                   6:  (* order finished *)
                       IF #sRecv.Echo.Start AND #sRecv.ErrorCode <> 16#FFFF THEN
                           #sSend.Start := FALSE;
                           #sHelp.EnableTime := FALSE;
                           IF #sRecv.ErrorCode = 16#0000 THEN
                               #sHelp.Step[#tIndex] := #sHelp.Step[#tIndex] + 1;
                           ELSE
                               #oErrorCode := 203;
                               #sHelp.Step[#tIndex] := 698;
                           END_IF;
                       ELSIF #sHelp.Abort THEN
                           #sHelp.Step[#tIndex] := 10;
                       ELSE
                           #sHelp.EnableTime := TRUE;
                           IF #sHelp.CmdTimer.Q THEN
                               #oErrorCode := 204;
                               #sHelp.Step[#tIndex] := 699;
                           END_IF;
                       END_IF;

                   7:  (* start order *)
                       IF (#sRecv.Echo.Status = 16#0000) AND #sRecv.CycleEnd THEN
                           #sSend.ReadLastResult := TRUE;
                           #sHelp.EnableTime := FALSE;
                           #sHelp.Step[#tIndex] := #sHelp.Step[#tIndex] + 1;
                       END_IF;

                   8:  (* order accepted *)
                       IF #sRecv.Echo.ReadLastResult AND #sRecv.ErrorCode = 16#FFFF THEN
                           #sHelp.EnableTime := FALSE;
                           #sHelp.Step[#tIndex] := #sHelp.Step[#tIndex] + 1;
                       ELSE
                           #sHelp.EnableTime := TRUE;
                           IF #sHelp.CmdTimer.Q THEN
                               #oErrorCode := 204;
                               #sHelp.Step[#tIndex] := 899;
                           END_IF;
                       END_IF;

                   9:  (* order finished *)
                       IF #sRecv.Echo.ReadLastResult AND #sRecv.ErrorCode <> 16#FFFF THEN
                           #sSend.ReadLastResult := FALSE;
                           #sHelp.EnableTime := FALSE;
                           IF #sRecv.ErrorCode = 16#0000 THEN
                               #sHelp.Step[#tIndex] := 997;
                           ELSE
                               #oErrorCode := 203;
                               #sHelp.Step[#tIndex] := 998;
                           END_IF;
                       ELSE
                           #sHelp.EnableTime := TRUE;
                           IF #sHelp.CmdTimer.Q THEN
                               #oErrorCode := 204;
                               #sHelp.Step[#tIndex] := 999;
                           END_IF;
                       END_IF;

                   10:  (* abort order *)
                       #sHelp.Step[#tIndex] := 1099;

                   299,398,399,599,698,699,899,997,998,999,1099:
                       #sSend.Reset := FALSE;
                       #sSend.Start := FALSE;
                       #sSend.ReadLastResult := FALSE;
                       #sHelp.MeasureAct := FALSE;
                       #sHMI.Trigger.Measure := FALSE;
                       #sHelp.Abort := FALSE;
                       IF #oErrorCode = 0 THEN
                           #oResult := #sRecv.Result;
                           #oMeasureOk := TRUE;
                       END_IF;
               END_CASE;
           END_IF;
       END_REGION

       (* update outputs *)
       #oDeviceReady := #sRecv.CycleEnd;
       #oPressure.Value := UDINT_TO_REAL(#sRecv.ActPressure) / 1000.0;
       CASE #sRecv.PressureUnitCode OF
           0000:
               #oPressure.Unit := 'cm3/s';
           1000:
               #oPressure.Unit := 'cm3/min';
           2000:
               #oPressure.Unit := 'cm3/h';
           3000:
               #oPressure.Unit := 'mm3/h';
           4000:
               #oPressure.Unit := 'Pa';
           5000:
               #oPressure.Unit := 'Pa/s';
           6000:
               #oPressure.Unit := 'Pa';
           7000:
               #oPressure.Unit := 'Pa';
           8000:
               #oPressure.Unit := 'Pa/s';
           9000:
               #oPressure.Unit := 'Pa/s';
           11000:
               #oPressure.Unit := 'bar';
           12000:
               #oPressure.Unit := 'KPa';
           13000:
               #oPressure.Unit := 'psi';
           14000:
               #oPressure.Unit := 'mbar';
           15000:
               #oPressure.Unit := 'MPa';
           43000:
               #oPressure.Unit := 'Pa';
           44000:
               #oPressure.Unit := 'Pa';
           45000:
               #oPressure.Unit := 'Pa/s';
           46000:
               #oPressure.Unit := 'In3/s';
           47000:
               #oPressure.Unit := 'In3/min';
           48000:
               #oPressure.Unit := 'In3/h';
           49000:
               #oPressure.Unit := 'Ft3/h';
           50000:
               #oPressure.Unit := 'mL/s';
           51000:
               #oPressure.Unit := 'mL/min';
           52000:
               #oPressure.Unit := 'mL/h';
           58000:
               #oPressure.Unit := 'cm3/s';
           59000:
               #oPressure.Unit := 'cm3/min';
           60000:
               #oPressure.Unit := 'cm3/h';
           76000:
               #oPressure.Unit := 'Ft3/s';
           77000:
               #oPressure.Unit := 'Ft3/min';
           84000:
               #oPressure.Unit := 'sccm';
           ELSE
               ;
       END_CASE;
       #oActProgStep := #sRecv.ActProgStep;
       #oActProgNo := #sRecv.ActProgram + 1;

       (* update hmi *)
       #sHMI.Status.DeviceReady := #oDeviceReady;
       #sHMI.Status.Ready := #oReady;
       #sHMI.Status.Error := #oError;
       #sHMI.Status.SetProgOk := #oSetProgOk;
       #sHMI.Status.MeasureOk := #oMeasureOk;
       #sHMI.Status.ErrorCode := #oErrorCode;
       #sHMI.Status.Result := #oResult;
       #sHMI.Status.Pressure := #oPressure;
       #sHMI.Status.ActProgStep := #oActProgStep;
       #sHMI.Status.ActProgNo := #oActProgNo;
       #sHMI.Status.ElapsedTime := #oElapsedTime;

       (* set ready for command flag *)
       IF (#oErrorCode = 0) AND (#sHelp.OrderCnt = 0) AND #oDeviceReady AND NOT #sHelp.SetProgAct AND NOT #sHelp.MeasureAct THEN
           #oReady := TRUE;
       ELSE
           #oReady := FALSE;
       END_IF;

       (* move static bits to output bytes *)
       #sArrayOutput[1, 1].%X0 := #sSend.Reset;
       #sArrayOutput[1, 1].%X1 := #sSend.Start;
       #sArrayOutput[1, 1].%X2 := #sSend.StartSpec;
       #sArrayOutput[1, 1].%X3 := #sSend.ProgramSel AND "ClockMemory0.8s";
       #sArrayOutput[1, 1].%X5 := #sSend.ReadPara ;
       #sArrayOutput[1, 2].%X7 := #sSend.ReadLastResult AND "ClockMemory0.8s";
       #sArrayOutput[1, 7] := #sSend.ProgNo.%B0;
       REGION SpecialCycle
           // Statement section REGION
           IF NOT #ioSpecialCycle THEN
               #SpecialCycleStep := 0;
           END_IF;
           IF #ioSpecialCycle AND #SpecialCycleStep = 0 AND #oReady AND #oDeviceReady THEN
               #SpecialCycleStep := 10;
           END_IF;
           #IEC_Timer_0_Instance(IN := #SpecialCycleStep = 10,
                                 PT := t#0.2s);
           #IEC_Timer_1_Instance(IN := #SpecialCycleStep = 20,
                                 PT := t#0.4s);
           CASE #SpecialCycleStep OF
               10://标志清零
                   #sHelp.EnableTime := FALSE;
                   #sArrayOutput[1, 9] := 16#00;
                   #sArrayOutput[1, 10] := 16#00;
                   IF #IEC_Timer_0_Instance.Q THEN
                       #SpecialCycleStep := 20;
                   END_IF;
               20://赋值
                   #sHelp.EnableTime := FALSE;
                   #sArrayOutput[1, 9] := 16#08;
                   #sArrayOutput[1, 10] := 16#00;
                   #sSend.StartSpec := 1;
                   IF #IEC_Timer_1_Instance.Q THEN
                       #SpecialCycleStep := 30;
                   END_IF;

               30://触发
                   #sHelp.EnableTime := FALSE;
                   #sSend.Start := 1;
                   #SpecialCycleStep := 40;
               40://运行
                   IF #sRecv.Echo.StartSpec THEN
                       #sHelp.EnableTime := FALSE;
                       #SpecialCycleStep := 50;
                   END_IF;
                   #sHelp.EnableTime := TRUE;
                   IF #sHelp.CmdTimer.Q THEN
                       #oErrorCode := 1004;
                       #SpecialCycleStep := 99;
                   END_IF;
               50://完成
                   IF NOT #oReady AND NOT #oDeviceReady THEN
                       #sHelp.EnableTime := FALSE;
                       #sSend.Start := #sSend.StartSpec := 0;
                       #SpecialCycleStep := 60;
                   END_IF;
                   #sHelp.EnableTime := TRUE;
                   IF #sHelp.CmdTimer.Q THEN
                       #oErrorCode := 1005;
                       #SpecialCycleStep := 99;
                   END_IF;
               60://完成
                   IF #oReady AND #oDeviceReady THEN
                       #ioSpecialCycle := #sSend.StartSpec := 0;
                       #sHelp.EnableTime := FALSE;
                   END_IF;
               99:
                   #sSend.Start := #sSend.StartSpec := 0;
                   #ioSpecialCycle := 0;
           END_CASE;

       END_REGION
       REGION ReadProTime
           // Statement section REGION
           IF NOT #ioReadProTime THEN
               #ReadProTimeStep := 0;
           END_IF;
           IF #ioReadProTime AND #ReadProTimeStep = 0 AND #oReady AND #oDeviceReady THEN
               #ReadProTimeStep := 10;
           END_IF;
           #IEC_Timer_0_Instance_1(IN := #ReadProTimeStep = 20,
                                 PT := t#0.1s);
         #IEC_Timer_1_Instance_1(IN := #ReadProTimeStep = 20,
                                 PT := t#0.3s);

           CASE #ReadProTimeStep OF
               10://标志
                   #sHelp.EnableTime := FALSE;
                   #sArrayOutput[1, 33] := 16#04;
                   #sArrayOutput[1, 34] := 16#00;
                   #sArrayOutput[1, 35] := 16#01;
                   #sArrayOutput[1, 36] := 16#00;
                   #sArrayOutput[1, 37] := 16#02;
                   #sArrayOutput[1, 38] := 16#00;
                   #sArrayOutput[1, 39] := 16#03;
                   #sArrayOutput[1, 40] := 16#00;
                   #sArrayOutput[1, 41] := 16#09;
                   #sArrayOutput[1, 42] := 16#00;
                   #ReadProTimeStep := 20;

               20://赋值
                   #sHelp.EnableTime := FALSE;
                   #sArrayOutput[1, 33] := 16#04;
                   #sArrayOutput[1, 34] := 16#00;
                   #sArrayOutput[1, 35] := 16#01;
                   #sArrayOutput[1, 36] := 16#00;
                   #sArrayOutput[1, 37] := 16#02;
                   #sArrayOutput[1, 38] := 16#00;
                   #sArrayOutput[1, 39] := 16#03;
                   #sArrayOutput[1, 40] := 16#00;
                   #sArrayOutput[1, 41] := 16#09;
                   #sArrayOutput[1, 42] := 16#00;

                   IF #IEC_Timer_0_Instance_1.Q THEN
                       #sSend.ReadPara := 1;
                   END_IF;
                   IF  #sRecv.Echo.ReadPara OR #IEC_Timer_1_Instance_1.Q THEN
                       #ReadProTimeStep := 30;
                   END_IF;
               30://触发
                   #sHelp.EnableTime := FALSE;

                   #ReadProTimeStep := 40;
               40://运行
                   #ReadProTimeStep := 50;
                   #sHelp.EnableTime := TRUE;
                   IF #sHelp.CmdTimer.Q THEN 
                       #oErrorCode := 1004;
                       #ReadProTimeStep := 99;
                   END_IF;
               50://完成
                   #ReadProTimeStep := 60;

               60://完成
                   IF #oReady AND #oDeviceReady THEN
                       #ioReadProTime := #sSend.ReadPara := 0;
                       #sHelp.EnableTime := FALSE;
                   END_IF;
               99:
                   #sSend.Start := #sSend.ReadPara := 0;
                   #ioReadProTime := 0;
           END_CASE;

       END_REGION


       (* Cyclic write plc output to tester input *)
       #tRetval.DPWR[1] := DPWR_DAT(LADDR := #iHWID_Slot5,
                                    RECORD := #sArrayOutput[1]);
       #tRetval.DPWR[2] := DPWR_DAT(LADDR := #iHWID_Slot6,
                                    RECORD := #sArrayOutput[2]);
       #tRetval.DPWR[3] := DPWR_DAT(LADDR := #iHWID_Slot7,
                                    RECORD := #sArrayOutput[3]);
       #tRetval.DPWR[4] := DPWR_DAT(LADDR := #iHWID_Slot8,
                                    RECORD := #sArrayOutput[4]);
       IF #tRetval.DPWR[1] <> 0 OR
           #tRetval.DPWR[2] <> 0 OR
           #tRetval.DPWR[3] <> 0 OR
           #tRetval.DPWR[4] <> 0  THEN
           #oErrorCode := 101; // Error cyclic write
       END_IF;

       (* handle errors within block *)
       #tRetval.LocallyErrID := GET_ERR_ID();
       IF #tRetval.LocallyErrID <> 0 THEN
           (* reset fieldbus output *)
           FOR #tLoop := 1 TO UINT_TO_INT(#cSlotAmount) DO
               UFILL_BLK(IN := 0,
                         COUNT := #cFieldbusBytes,
                         OUT => #sArrayOutput[#tLoop, 01]);
           END_FOR;
           #oErrorCode := 102; // Error within block
       END_IF;

   END_IF;
END_FUNCTION_BLOCK

FUNCTION_BLOCK "FB_Analog"   // FB4090, LAD
{ S7_Optimized_Access := 'TRUE' }
// stored: AutoNumber false, MemoryReserve 100, SetENOAutomatically false
   VAR_INPUT
      iSysInface : "RCS_SysComInterface_V1";
      "iunit in" : UInt;   // 0:mA(电流);1:V(电压)
      "iunit out" : UInt;   // 0:mm(毫米);1:N(牛顿);2.KN(千牛顿);3.bar(帕);4:kPa;5:mbar;6:bar;7:m/s;8:°
      "iHardware input" : Word;   // 硬件输入
      iRangeDown : Real;
      iRangeUp : Real;
   END_VAR
   VAR_IN_OUT
      io_Dev : "ST_GeneralAnalog";
   END_VAR
   VAR_TEMP
      TmpMidReal0 : Real;
   END_VAR
BEGIN

REGION Network 1: 启动条件 / Starting condition
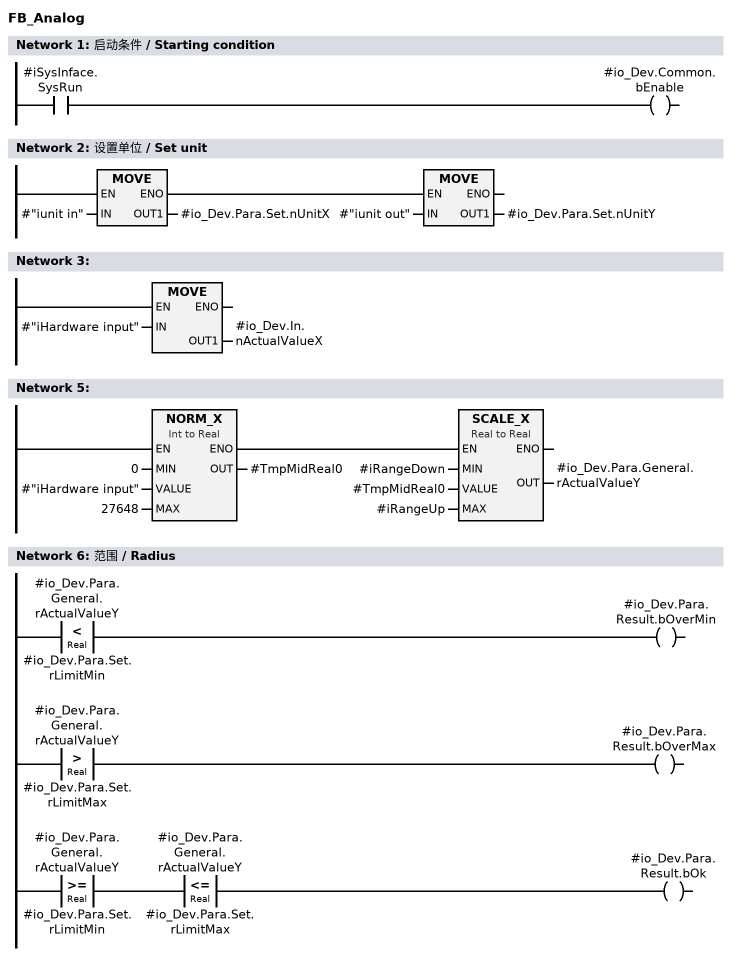
   RUNG wire#powerrail
      Contact( #iSysInface.SysRun )
      Coil( #io_Dev.Common.bEnable )
   END_RUNG
   // the same network as SCL:
   #io_Dev.Common.bEnable := #iSysInface.SysRun;
END_REGION

REGION Network 2: 设置单位 / Set unit
   RUNG wire#powerrail
      Move(in := #"iunit in", out1 => #io_Dev.Para.Set.nUnitX)
      Move(in := #"iunit out", out1 => #io_Dev.Para.Set.nUnitY)
   END_RUNG
   // the same network as SCL:
   #io_Dev.Para.Set.nUnitX := #"iunit in";
   #io_Dev.Para.Set.nUnitY := #"iunit out";
END_REGION

REGION Network 3
   RUNG wire#powerrail
      Move(in := #"iHardware input", out1 => #io_Dev.In.nActualValueX)
   END_RUNG
   // the same network as SCL:
   #io_Dev.In.nActualValueX := #"iHardware input";
END_REGION

REGION Network 5
   RUNG wire#powerrail
      { S7_Templates := "[SrcType := Int, DestType := Real]" } Normalize(min := 0, value := #"iHardware input", max := 27648, out => #TmpMidReal0)
      { S7_Templates := "[SrcType := Real, DestType := Real]" } Scale(min := #iRangeDown, value := #TmpMidReal0, max := #iRangeUp, out => #io_Dev.Para.General.rActualValueY)
   END_RUNG
   // the same network as SCL:
   #TmpMidReal0 := NORM_X(MIN := 0, VALUE := #"iHardware input", MAX := 27648);
   #io_Dev.Para.General.rActualValueY := SCALE_X(MIN := #iRangeDown, VALUE := #TmpMidReal0, MAX := #iRangeUp);
END_REGION

REGION Network 6: 范围 / Radius
   RUNG wire#powerrail
      { S7_Templates := "SrcType := Real" } LT_Contact(in1 := #io_Dev.Para.General.rActualValueY, in2 := #io_Dev.Para.Set.rLimitMin)
      Coil( #io_Dev.Para.Result.bOverMin )
   END_RUNG
   RUNG wire#powerrail
      { S7_Templates := "SrcType := Real" } GT_Contact(in1 := #io_Dev.Para.General.rActualValueY, in2 := #io_Dev.Para.Set.rLimitMax)
      Coil( #io_Dev.Para.Result.bOverMax )
   END_RUNG
   RUNG wire#powerrail
      { S7_Templates := "SrcType := Real" } GE_Contact(in1 := #io_Dev.Para.General.rActualValueY, in2 := #io_Dev.Para.Set.rLimitMin)
      { S7_Templates := "SrcType := Real" } LE_Contact(in1 := #io_Dev.Para.General.rActualValueY, in2 := #io_Dev.Para.Set.rLimitMax)
      Coil( #io_Dev.Para.Result.bOk )
   END_RUNG
   // the same network as SCL:
   #io_Dev.Para.Result.bOverMin := #io_Dev.Para.General.rActualValueY < #io_Dev.Para.Set.rLimitMin;
   #io_Dev.Para.Result.bOverMax := #io_Dev.Para.General.rActualValueY > #io_Dev.Para.Set.rLimitMax;
   #io_Dev.Para.Result.bOk := (#io_Dev.Para.General.rActualValueY >= #io_Dev.Para.Set.rLimitMin) AND (#io_Dev.Para.General.rActualValueY <= #io_Dev.Para.Set.rLimitMax);
END_REGION
END_FUNCTION_BLOCK

FUNCTION_BLOCK "FB_Keyence_SR1000"   // FB1230, SCL
{ S7_Optimized_Access := 'TRUE' }
// stored: AutoNumber false, MemoryReserve 100, SetENOAutomatically false
   VAR_INPUT
      "I_Handshake and Genera_InAdr" : HW_IO;
      I_BUSYStatusBits_InAdr : HW_IO;
      I_CompletionStatus_InAdr : HW_IO;
      I_ErrorStatusBits_InAdr : HW_IO;
      "I_Terminal Status InAdr" : HW_IO;
      "I_Unstable Read Status Bits_InAdr" : HW_IO;
      "I_Matching Level and Total_InAdr" : HW_IO;
      "I_Operation Result Status InAdr" : HW_IO;
      "I_Read Data 128Byte InAdr" : HW_IO;
      "I_Latch and Error OutAdr" : HW_IO;
      "I_Operation instruction_OutAdr" : HW_IO;
      "I_Completion OutAdr" : HW_IO;
      "I_Parameter Bank Number_OutAdr" : HW_IO;
      "I_User Data 128Byte_OutAdr" : HW_IO;
   END_VAR
   VAR_OUTPUT
      io_nError : Int;
      io_nWarning : Int;
   END_VAR
   VAR_IN_OUT
      IO_udtData : "ST_KeyenceSR1000";
   END_VAR
   VAR
      s_nValue : Array[0..20] of Int;
      sUP : Array[0..10] of R_TRIG;
      TON { S7_SetPoint := 'True'} : Array[0..10] of TON_TIME;
      FB_Step { S7_SetPoint := 'True'} : "FB_Step";
      sPN_IN : Struct
         Handshake : Byte;
         BUSYStatusBits : Byte;
         CompletionStatus : Byte;
         ErrorStatusBits : Byte;
         TerminalStatus : Byte;
         UnstableReadStatusBits : Byte;
         MatchingLevelandTotal : Array[1..8] of Byte;
         OperationResultStatus : Array[1..20] of Byte;
         ReadData128Byte : Array[1..136] of Byte;
      END_STRUCT;
      sPN_Out : Struct
         LatchErrorClear : Byte;   // Latch and Error Clear Control Bits
         OperationInstruction : Byte;   // Operation instruction Control Bits
         Completion : Byte;   // Completion Clear Control Bits
         ParBankNo : Array[1..2] of Byte;   // Parameter Bank Number
         UserData128byte : Array[1..136] of Byte;   // UserData128byte
      END_STRUCT;
      Flag : Array[0..10] of Bool;
   END_VAR
   VAR_TEMP
      tInt : Array[1..8] of Int;
      i : Int;
      TempBytes : Array[1..128] of Char;
   END_VAR
BEGIN
   REGION Read PN Data 读取PN数据
       // 插槽1
       #s_nValue[1] := DPRD_DAT(LADDR := #"I_Handshake and Genera_InAdr",
                                RECORD => #sPN_IN.Handshake);
       //插槽2
       #s_nValue[2] := DPRD_DAT(LADDR := #I_BUSYStatusBits_InAdr,
                                RECORD => #sPN_IN.BUSYStatusBits);
       //插槽3
       #s_nValue[3] := DPRD_DAT(LADDR := #I_CompletionStatus_InAdr,
                                RECORD => #sPN_IN.CompletionStatus);
       //插槽4
       #s_nValue[4] := DPRD_DAT(LADDR := #I_ErrorStatusBits_InAdr,
                                RECORD => #sPN_IN.ErrorStatusBits);
       //插槽5
       #s_nValue[5] := DPRD_DAT(LADDR := #"I_Terminal Status InAdr",
                                RECORD => #sPN_IN.TerminalStatus);
       //插槽6
       #s_nValue[6] := DPRD_DAT(LADDR := #"I_Unstable Read Status Bits_InAdr",
                                RECORD => #sPN_IN.UnstableReadStatusBits);
       //插槽7
       #s_nValue[7] := DPRD_DAT(LADDR := #"I_Matching Level and Total_InAdr",
                                RECORD => #sPN_IN.MatchingLevelandTotal);
       //插槽8
       #s_nValue[8] := DPRD_DAT(LADDR := #"I_Operation Result Status InAdr",
                                RECORD => #sPN_IN.OperationResultStatus);
       //插槽9
       #s_nValue[9] := DPRD_DAT(LADDR := #"I_Read Data 128Byte InAdr",
                                RECORD => #sPN_IN.ReadData128Byte);

   END_REGION

   REGION CopyReadData()
       //************************************************************************************************
       //分配输入数据(控制数据解析)/Asignment of the input data (control word)
       //************************************************************************************************
       #IO_udtData.In.bBusy := #sPN_IN.BUSYStatusBits.%X1;
       #IO_udtData.In.bError := #sPN_IN.Handshake.%X0;
       #IO_udtData.In.bReadComplete := #sPN_IN.CompletionStatus.%X0;
       #IO_udtData.In.bReadFailure := #sPN_IN.ErrorStatusBits.%X0;
       #IO_udtData.In.nReadResultCode := #sPN_IN.OperationResultStatus[4];

   END_REGION

   REGION Error Code 报错信息
       //流程超时/Process overtime alarm   X0
       #TON[1](IN := #IO_udtData.Common.nMode <> 0,
               PT := T#12S);
       IF #TON[1].Q THEN
           #IO_udtData.Common.nErrorNo := 1;
           #io_nError.%X0 := 1;
       END_IF;

       //读码超时

       #TON[2](IN := NOT #FB_Step.sCondition AND #FB_Step.sNextNo = 1100,
               PT := T#8S);

       //错误标志/Error flag
       //
       IF #IO_udtData.Common.nErrorNo <> 0 THEN
           #IO_udtData.Common.bError := TRUE;
           #IO_udtData.Common.nMode := 0;
       END_IF;

       //复位报警信息/Reset alarm messages
       IF #IO_udtData.Common.bReset AND #IO_udtData.Common.bError THEN
           #IO_udtData.Common.nErrorNo := 0;
           #io_nError := 0;
           #IO_udtData.Common.bError := FALSE;
       END_IF;
       //报警复位
       #IO_udtData.Out.bErrorClear := #IO_udtData.Common.bReset;

   END_REGION

   REGION 提示信息
       // Statement section REGION
       #IO_udtData.Common.nWarningNo := #IO_udtData.In.nReadResultCode;
   END_REGION


   REGION Data 读码数据解析
       IF #IO_udtData.In.bReadComplete THEN
           #IO_udtData.In.nDataSize := #sPN_IN.ReadData128Byte[8] - 1;
           FOR #i := 1 TO 128 DO
               #IO_udtData.In.aData[#i] := #sPN_IN.ReadData128Byte[#i + 8];
           END_FOR;
           Chars_TO_Strg(Chars := #IO_udtData.In.aData,
                         pChars := 0,
                         Cnt := #IO_udtData.In.nDataSize,
                         Strg => #IO_udtData.RecordCode);
       END_IF;
   END_REGION

   REGION AutoStep
       #FB_Step(1);
       IF #IO_udtData.Common.nMode <> 0 THEN
           CASE #FB_Step.sCurrNo OF
               0:
                   #FB_Step.sCondition := #IO_udtData.Common.nMode = 1;
                   #FB_Step.sNextNo := 1000;
               1000://开始读取
                   IF #FB_Step.sPls THEN
                       #IO_udtData.Out.bReadRequest := 1;
                       #IO_udtData.RecordCode := '';
                       #IO_udtData.In.aData := #TempBytes;
                       #IO_udtData.In.nDataSize := 0;
                       #IO_udtData.Common.bDone := 0;
                       #IO_udtData.Common.bNG := 0;
                       #IO_udtData.Common.bOK := 0;
                   END_IF;
                   #FB_Step.sCondition := #IO_udtData.In.bBusy;
                   #FB_Step.sNextNo := 1100;
               1100://等待读取完成

                   #FB_Step.sDealyTime := T#10MS;

                   #FB_Step.sCondition :=( #IO_udtData.In.bReadComplete AND NOT #IO_udtData.In.bBusy ) OR #TON[2].Q;
                   IF #FB_Step.sCondition THEN
                       #IO_udtData.Out.bReadRequest := 0;
                   END_IF;
                   #FB_Step.sNextNo := 1200;
               1200://判断读取结果
                   IF #IO_udtData.RecordCode = 'ERROR' THEN
                       #IO_udtData.Common.bNG := 1;//读取NG
                       #IO_udtData.Common.bOK := 0;
                   ELSE
                       #IO_udtData.Common.bNG := 0;
                       #IO_udtData.Common.bOK := 1;//读取OK
                   END_IF;
                   #FB_Step.sCondition := 1;
                   #FB_Step.sNextNo := 1300;
               1300://读取完成
                   IF #FB_Step.sPls THEN
                       #IO_udtData.Out.bReadComlpleteClear := 1;
                   END_IF;
                   #FB_Step.sCondition := NOT #IO_udtData.In.bReadComplete AND NOT #IO_udtData.In.bReadFailure;
                   #FB_Step.sNextNo := 1400;
               1400://
                   IF #FB_Step.sPls THEN
                       #IO_udtData.Out.bReadComlpleteClear := 0;
                       #IO_udtData.Common.bDone := 1;
                       #IO_udtData.Common.nMode := 0;
                   END_IF;
                   #FB_Step.sCondition := 1;
                   #FB_Step.sNextNo := 0;
           END_CASE;
       ELSE
           #FB_Step.sCurrNo := 0;
           #IO_udtData.Out.bReadComlpleteClear := 0;
           #IO_udtData.Out.bReadRequest := 0;
       END_IF;
   END_REGION

   REGION CopyWriteData()   
       //************************************************************************************************
       //分配输出数据(控制数据解析)/Asignment of the output data (control word)
       //************************************************************************************************
       #sPN_Out.OperationInstruction.%X0 := #IO_udtData.Out.bReadRequest;
       #sPN_Out.LatchErrorClear.%X7:= #IO_udtData.Out.bErrorClear;
       #sPN_Out.Completion.%X0 := #IO_udtData.Out.bReadComlpleteClear;



   END_REGION

   REGION Write Data 写入PN数据
       // 插槽10
       #s_nValue[10] := DPWR_DAT(LADDR := #"I_Latch and Error OutAdr",
                                RECORD := #sPN_Out.LatchErrorClear);
       // 插槽11
       #s_nValue[11] := DPWR_DAT(LADDR := #"I_Operation instruction_OutAdr",
                                RECORD := #sPN_Out.OperationInstruction);
       //插槽12
      #s_nValue[12] := DPWR_DAT(LADDR := #"I_Completion OutAdr",
                                RECORD := #sPN_Out.Completion);
       // 插槽13
      #s_nValue[13] := DPWR_DAT(LADDR := #"I_Parameter Bank Number_OutAdr",
                                RECORD := #sPN_Out.ParBankNo);
       // 插槽14
       #s_nValue[14] := DPWR_DAT(LADDR := #"I_User Data 128Byte_OutAdr",
                                RECORD := #sPN_Out.UserData128byte);
   END_REGION
END_FUNCTION_BLOCK

FUNCTION_BLOCK "FB_Step"   // FB5002, LAD
{ S7_Optimized_Access := 'TRUE' }
// stored: AutoNumber false, MemoryReserve 100, SetENOAutomatically false
   VAR_INPUT
      I_bRun : Bool;   // 运行条件
   END_VAR
   VAR
      sCurrNo : UInt;   // 当前步号
      sNextNo : UInt;   // 下一步号
      sPls : Bool;   // 步序脉冲
      sCondition : Bool;   // 完成条件
      sRunJump : Bool;   // 与输入的运行条件并行
      sTON : TON_TIME;
      sDealyTime { S7_SetPoint := 'True'} : Time;
      sTempNo : UInt;
      bInitialization : Bool;   // 初始化
   END_VAR
   VAR_TEMP   // added for the SCL form of the ladder/FBD networks
      _w1 : Bool;
   END_VAR
BEGIN

REGION Network 1
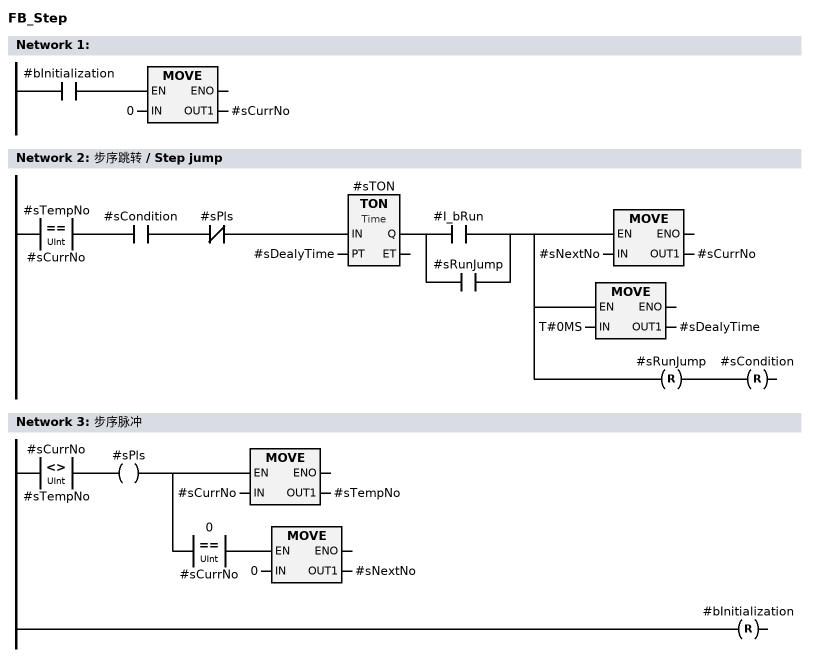
   RUNG wire#powerrail
      Contact( #bInitialization )
      Move(in := 0, out1 => #sCurrNo)
   END_RUNG
   // the same network as SCL:
   IF #bInitialization THEN #sCurrNo := 0; END_IF;
END_REGION

REGION Network 2: 步序跳转 / Step jump
   RUNG wire#powerrail
      { S7_Templates := "SrcType := UInt" } EQ_Contact(in1 := #sTempNo, in2 := #sCurrNo)
      Contact( #sCondition )
      I_Contact( #sPls )
      { S7_Templates := "time_type := Time" } #sTON.TON(pt := #sDealyTime, et =>)
      wire#w1
      Contact( #I_bRun )
      wire#w2
      Move(in := #sNextNo, out1 => #sCurrNo)
   END_RUNG
   RUNG wire#w1
      Contact( #sRunJump )
   END_RUNG wire#w2
   RUNG wire#w2
      Move(in := T#0MS, out1 => #sDealyTime)
   END_RUNG
   RUNG wire#w2
      R_Coil( #sRunJump )
      R_Coil( #sCondition )
   END_RUNG
   // the same network as SCL:
   #sTON(IN := (#sTempNo = #sCurrNo) AND #sCondition AND NOT #sPls, PT := #sDealyTime);   // TON
   IF #sTON.Q AND (#I_bRun OR #sRunJump) THEN
       #sCurrNo := #sNextNo;
       #sDealyTime := T#0MS;
   END_IF;
   #_w1 := #sTON.Q AND (#I_bRun OR #sRunJump);
   IF #_w1 THEN
       #sRunJump := FALSE;
       #sCondition := FALSE;
   END_IF;
END_REGION

REGION Network 3: 步序脉冲
   RUNG wire#powerrail
      { S7_Templates := "SrcType := UInt" } NE_Contact(in1 := #sCurrNo, in2 := #sTempNo)
      Coil( #sPls )
      wire#w1
      Move(in := #sCurrNo, out1 => #sTempNo)
   END_RUNG
   RUNG wire#w1
      { S7_Templates := "SrcType := UInt" } EQ_Contact(in1 := 0, in2 := #sCurrNo)
      Move(in := 0, out1 => #sNextNo)
   END_RUNG
   RUNG wire#powerrail
      R_Coil( #bInitialization )
   END_RUNG
   // the same network as SCL:
   #sPls := #sCurrNo <> #sTempNo;
   IF #sPls THEN #sTempNo := #sCurrNo; END_IF;
   IF #sPls AND (0 = #sCurrNo) THEN #sNextNo := 0; END_IF;
   #bInitialization := FALSE;
END_REGION
END_FUNCTION_BLOCK

FUNCTION "ST10Cyl_interface91-100" : Void   // FC1029, LAD
{ S7_Optimized_Access := 'FALSE' }
// stored: AutoNumber false, SetENOAutomatically false
   VAR_INPUT
      AlwaysON : Bool;
      E_stop : Bool;
   END_VAR
   VAR_TEMP
      tTest : Bool;
   END_VAR
BEGIN

REGION Network 1 (SCL): Cylinder 91-100 IO Interface (SCL)
END_REGION

REGION Network 2: CY91 interface
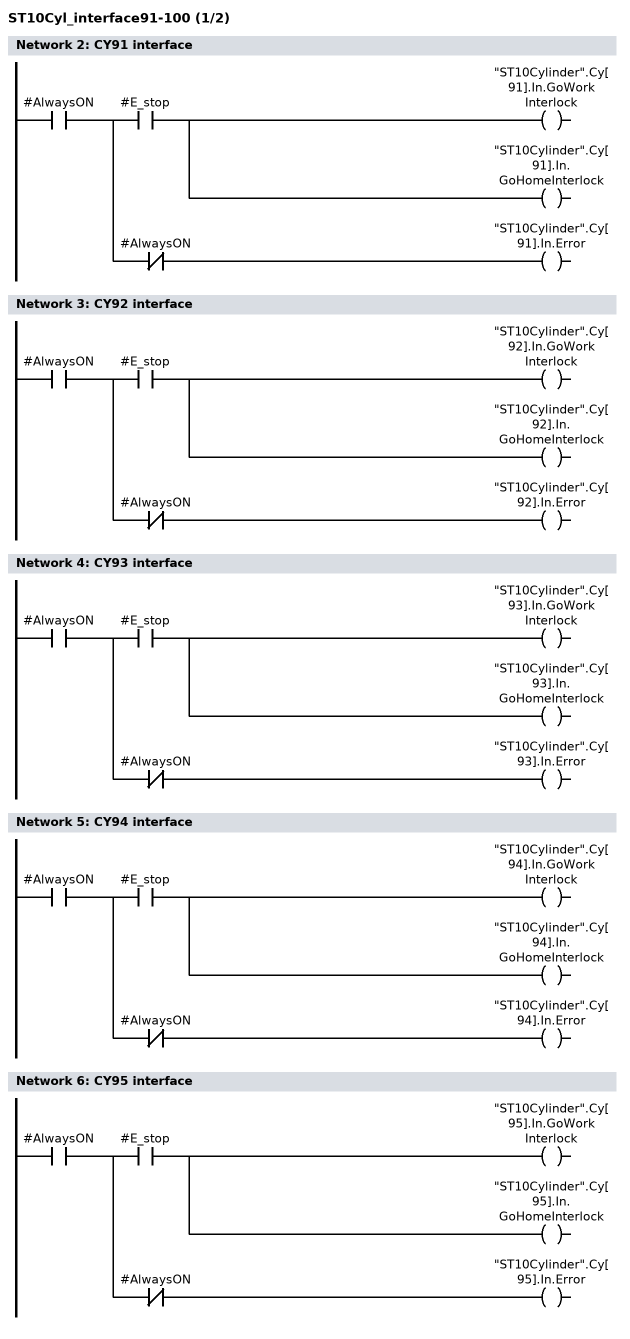
   RUNG wire#powerrail
      Contact( #AlwaysON )
      wire#w1
      Contact( #E_stop )
      wire#w2
      Coil( "ST10Cylinder".Cy[91].In.GoWorkInterlock )
   END_RUNG
   RUNG wire#w2
      Coil( "ST10Cylinder".Cy[91].In.GoHomeInterlock )
   END_RUNG
   RUNG wire#w1
      I_Contact( #AlwaysON )
      Coil( "ST10Cylinder".Cy[91].In.Error )
   END_RUNG
   // the same network as SCL:
   "ST10Cylinder".Cy[91].In.GoWorkInterlock := #AlwaysON AND #E_stop;
   "ST10Cylinder".Cy[91].In.GoHomeInterlock := #AlwaysON AND #E_stop;
   "ST10Cylinder".Cy[91].In.Error := #AlwaysON AND NOT #AlwaysON;
END_REGION

REGION Network 3: CY92 interface
   RUNG wire#powerrail
      Contact( #AlwaysON )
      wire#w1
      Contact( #E_stop )
      wire#w2
      Coil( "ST10Cylinder".Cy[92].In.GoWorkInterlock )
   END_RUNG
   RUNG wire#w2
      Coil( "ST10Cylinder".Cy[92].In.GoHomeInterlock )
   END_RUNG
   RUNG wire#w1
      I_Contact( #AlwaysON )
      Coil( "ST10Cylinder".Cy[92].In.Error )
   END_RUNG
   // the same network as SCL:
   "ST10Cylinder".Cy[92].In.GoWorkInterlock := #AlwaysON AND #E_stop;
   "ST10Cylinder".Cy[92].In.GoHomeInterlock := #AlwaysON AND #E_stop;
   "ST10Cylinder".Cy[92].In.Error := #AlwaysON AND NOT #AlwaysON;
END_REGION

REGION Network 4: CY93 interface
   RUNG wire#powerrail
      Contact( #AlwaysON )
      wire#w1
      Contact( #E_stop )
      wire#w2
      Coil( "ST10Cylinder".Cy[93].In.GoWorkInterlock )
   END_RUNG
   RUNG wire#w2
      Coil( "ST10Cylinder".Cy[93].In.GoHomeInterlock )
   END_RUNG
   RUNG wire#w1
      I_Contact( #AlwaysON )
      Coil( "ST10Cylinder".Cy[93].In.Error )
   END_RUNG
   // the same network as SCL:
   "ST10Cylinder".Cy[93].In.GoWorkInterlock := #AlwaysON AND #E_stop;
   "ST10Cylinder".Cy[93].In.GoHomeInterlock := #AlwaysON AND #E_stop;
   "ST10Cylinder".Cy[93].In.Error := #AlwaysON AND NOT #AlwaysON;
END_REGION

REGION Network 5: CY94 interface
   RUNG wire#powerrail
      Contact( #AlwaysON )
      wire#w1
      Contact( #E_stop )
      wire#w2
      Coil( "ST10Cylinder".Cy[94].In.GoWorkInterlock )
   END_RUNG
   RUNG wire#w2
      Coil( "ST10Cylinder".Cy[94].In.GoHomeInterlock )
   END_RUNG
   RUNG wire#w1
      I_Contact( #AlwaysON )
      Coil( "ST10Cylinder".Cy[94].In.Error )
   END_RUNG
   // the same network as SCL:
   "ST10Cylinder".Cy[94].In.GoWorkInterlock := #AlwaysON AND #E_stop;
   "ST10Cylinder".Cy[94].In.GoHomeInterlock := #AlwaysON AND #E_stop;
   "ST10Cylinder".Cy[94].In.Error := #AlwaysON AND NOT #AlwaysON;
END_REGION

REGION Network 6: CY95 interface
   RUNG wire#powerrail
      Contact( #AlwaysON )
      wire#w1
      Contact( #E_stop )
      wire#w2
      Coil( "ST10Cylinder".Cy[95].In.GoWorkInterlock )
   END_RUNG
   RUNG wire#w2
      Coil( "ST10Cylinder".Cy[95].In.GoHomeInterlock )
   END_RUNG
   RUNG wire#w1
      I_Contact( #AlwaysON )
      Coil( "ST10Cylinder".Cy[95].In.Error )
   END_RUNG
   // the same network as SCL:
   "ST10Cylinder".Cy[95].In.GoWorkInterlock := #AlwaysON AND #E_stop;
   "ST10Cylinder".Cy[95].In.GoHomeInterlock := #AlwaysON AND #E_stop;
   "ST10Cylinder".Cy[95].In.Error := #AlwaysON AND NOT #AlwaysON;
END_REGION

REGION Network 7: CY96 interface
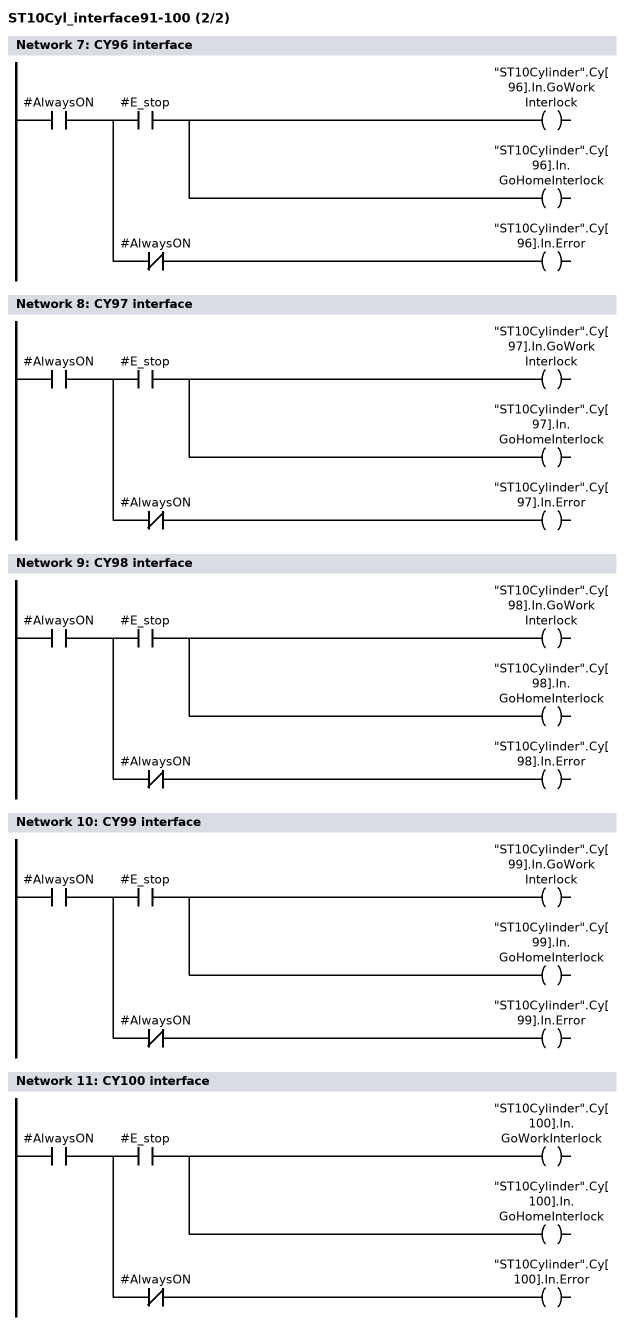
   RUNG wire#powerrail
      Contact( #AlwaysON )
      wire#w1
      Contact( #E_stop )
      wire#w2
      Coil( "ST10Cylinder".Cy[96].In.GoWorkInterlock )
   END_RUNG
   RUNG wire#w2
      Coil( "ST10Cylinder".Cy[96].In.GoHomeInterlock )
   END_RUNG
   RUNG wire#w1
      I_Contact( #AlwaysON )
      Coil( "ST10Cylinder".Cy[96].In.Error )
   END_RUNG
   // the same network as SCL:
   "ST10Cylinder".Cy[96].In.GoWorkInterlock := #AlwaysON AND #E_stop;
   "ST10Cylinder".Cy[96].In.GoHomeInterlock := #AlwaysON AND #E_stop;
   "ST10Cylinder".Cy[96].In.Error := #AlwaysON AND NOT #AlwaysON;
END_REGION

REGION Network 8: CY97 interface
   RUNG wire#powerrail
      Contact( #AlwaysON )
      wire#w1
      Contact( #E_stop )
      wire#w2
      Coil( "ST10Cylinder".Cy[97].In.GoWorkInterlock )
   END_RUNG
   RUNG wire#w2
      Coil( "ST10Cylinder".Cy[97].In.GoHomeInterlock )
   END_RUNG
   RUNG wire#w1
      I_Contact( #AlwaysON )
      Coil( "ST10Cylinder".Cy[97].In.Error )
   END_RUNG
   // the same network as SCL:
   "ST10Cylinder".Cy[97].In.GoWorkInterlock := #AlwaysON AND #E_stop;
   "ST10Cylinder".Cy[97].In.GoHomeInterlock := #AlwaysON AND #E_stop;
   "ST10Cylinder".Cy[97].In.Error := #AlwaysON AND NOT #AlwaysON;
END_REGION

REGION Network 9: CY98 interface
   RUNG wire#powerrail
      Contact( #AlwaysON )
      wire#w1
      Contact( #E_stop )
      wire#w2
      Coil( "ST10Cylinder".Cy[98].In.GoWorkInterlock )
   END_RUNG
   RUNG wire#w2
      Coil( "ST10Cylinder".Cy[98].In.GoHomeInterlock )
   END_RUNG
   RUNG wire#w1
      I_Contact( #AlwaysON )
      Coil( "ST10Cylinder".Cy[98].In.Error )
   END_RUNG
   // the same network as SCL:
   "ST10Cylinder".Cy[98].In.GoWorkInterlock := #AlwaysON AND #E_stop;
   "ST10Cylinder".Cy[98].In.GoHomeInterlock := #AlwaysON AND #E_stop;
   "ST10Cylinder".Cy[98].In.Error := #AlwaysON AND NOT #AlwaysON;
END_REGION

REGION Network 10: CY99 interface
   RUNG wire#powerrail
      Contact( #AlwaysON )
      wire#w1
      Contact( #E_stop )
      wire#w2
      Coil( "ST10Cylinder".Cy[99].In.GoWorkInterlock )
   END_RUNG
   RUNG wire#w2
      Coil( "ST10Cylinder".Cy[99].In.GoHomeInterlock )
   END_RUNG
   RUNG wire#w1
      I_Contact( #AlwaysON )
      Coil( "ST10Cylinder".Cy[99].In.Error )
   END_RUNG
   // the same network as SCL:
   "ST10Cylinder".Cy[99].In.GoWorkInterlock := #AlwaysON AND #E_stop;
   "ST10Cylinder".Cy[99].In.GoHomeInterlock := #AlwaysON AND #E_stop;
   "ST10Cylinder".Cy[99].In.Error := #AlwaysON AND NOT #AlwaysON;
END_REGION

REGION Network 11: CY100 interface
   RUNG wire#powerrail
      Contact( #AlwaysON )
      wire#w1
      Contact( #E_stop )
      wire#w2
      Coil( "ST10Cylinder".Cy[100].In.GoWorkInterlock )
   END_RUNG
   RUNG wire#w2
      Coil( "ST10Cylinder".Cy[100].In.GoHomeInterlock )
   END_RUNG
   RUNG wire#w1
      I_Contact( #AlwaysON )
      Coil( "ST10Cylinder".Cy[100].In.Error )
   END_RUNG
   // the same network as SCL:
   "ST10Cylinder".Cy[100].In.GoWorkInterlock := #AlwaysON AND #E_stop;
   "ST10Cylinder".Cy[100].In.GoHomeInterlock := #AlwaysON AND #E_stop;
   "ST10Cylinder".Cy[100].In.Error := #AlwaysON AND NOT #AlwaysON;
END_REGION
END_FUNCTION

FUNCTION_BLOCK "ST10_Stopper_FB"   // FB1160, LAD
{ S7_Optimized_Access := 'TRUE' }
// stored: AutoNumber false, MemoryReserve 100, SetENOAutomatically false
   VAR
      FB_Stopper_Instance { S7_SetPoint := 'True'} : Array[1..3] of "FB_Stopper";
   END_VAR
BEGIN

REGION Network 1 (SCL): A-托盘缓存阻挡气缸
       (*  
       REGION 允许释放条件,根据实际完善
           //马达运行中且工位一允许进料
           IF "ST350_Motor_InterfaceDB".aDev[1].Run  THEN
               "ST350_Stopper_InterfaceDB".Command[1].In.iReleaseClear := TRUE;
           ELSE
               "ST350_Stopper_InterfaceDB".Command[1].In.iReleaseClear := FALSE;
           END_IF;
       END_REGION

       REGION IO_image
           //InPut
           "ST350_Stopper_InterfaceDB".Command[1].In.iSensor := "iBurfferPalletDetection";//本站托盘到位
           "ST350_Stopper_InterfaceDB".Command[1].In.iNextSensor := "iWork01PalletDetection";//后站托盘到位
           "ST350_Stopper_InterfaceDB".Command[1].In.iNextValve := "oA-Lifting-01StopperCylinder";//后站挡停输出

           // //OutPut
            "ST10Cylinder".Cy[5].Inout.AutoGoWork:= "ST350_Stopper_InterfaceDB".Command[1].Out.oValve;//本站挡停输出
       END_REGION


       *)
END_REGION

REGION Network 2: #FB_Stopper_Instance[1] A-托盘缓存阻挡气缸
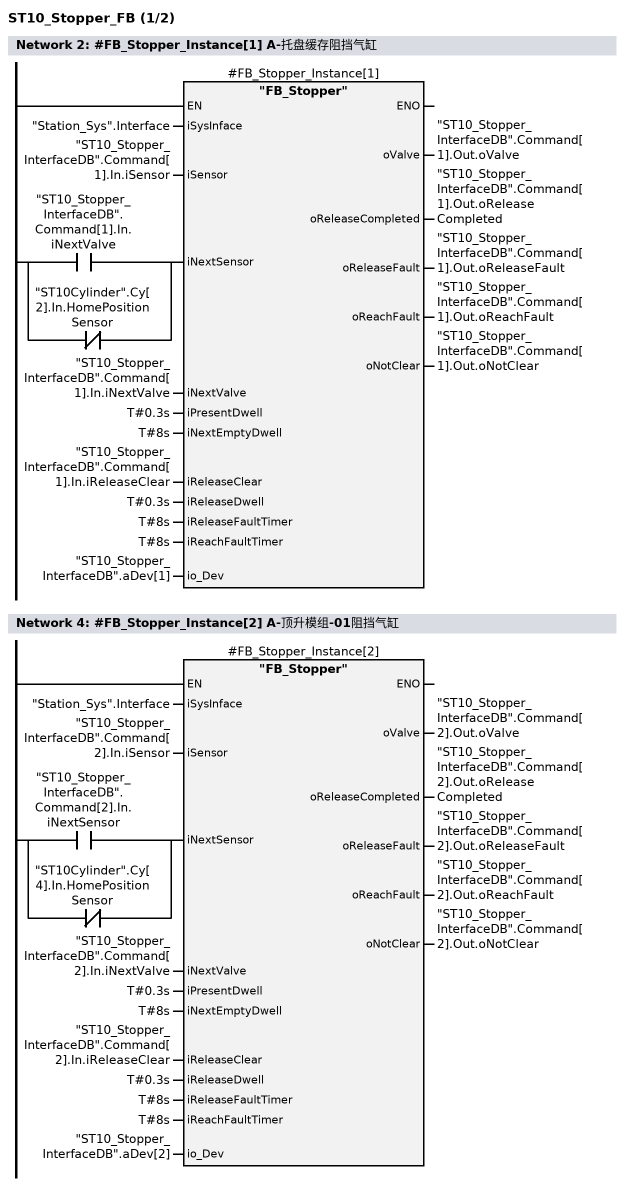
   RUNG wire#powerrail
      #FB_Stopper_Instance[1](iNextSensor := wire#w1, iSysInface := "Station_Sys".Interface, iSensor := "ST10_Stopper_InterfaceDB".Command[1].In.iSensor, iNextValve := "ST10_Stopper_InterfaceDB".Command[1].In.iNextValve, iPresentDwell := T#0.3s, iNextEmptyDwell := T#8s, iReleaseClear := "ST10_Stopper_InterfaceDB".Command[1].In.iReleaseClear, iReleaseDwell := T#0.3s, iReleaseFaultTimer := T#8s, iReachFaultTimer := T#8s, io_Dev := "ST10_Stopper_InterfaceDB".aDev[1], oValve => "ST10_Stopper_InterfaceDB".Command[1].Out.oValve, oReleaseCompleted => "ST10_Stopper_InterfaceDB".Command[1].Out.oReleaseCompleted, oReleaseFault => "ST10_Stopper_InterfaceDB".Command[1].Out.oReleaseFault, oReachFault => "ST10_Stopper_InterfaceDB".Command[1].Out.oReachFault, oNotClear => "ST10_Stopper_InterfaceDB".Command[1].Out.oNotClear)
   END_RUNG
   RUNG wire#powerrail
      Contact( "ST10_Stopper_InterfaceDB".Command[1].In.iNextValve )
   END_RUNG wire#w1
   RUNG wire#powerrail
      I_Contact( "ST10Cylinder".Cy[2].In.HomePositionSensor )
   END_RUNG wire#w1
   // the same network as SCL:
   #FB_Stopper_Instance[1](iSysInface := "Station_Sys".Interface,   // "FB_Stopper"
                           iSensor := "ST10_Stopper_InterfaceDB".Command[1].In.iSensor,
                           iNextSensor := "ST10_Stopper_InterfaceDB".Command[1].In.iNextValve OR NOT "ST10Cylinder".Cy[2].In.HomePositionSensor,
                           iNextValve := "ST10_Stopper_InterfaceDB".Command[1].In.iNextValve,
                           iPresentDwell := T#0.3s,
                           iNextEmptyDwell := T#8s,
                           iReleaseClear := "ST10_Stopper_InterfaceDB".Command[1].In.iReleaseClear,
                           iReleaseDwell := T#0.3s,
                           iReleaseFaultTimer := T#8s,
                           iReachFaultTimer := T#8s,
                           io_Dev := "ST10_Stopper_InterfaceDB".aDev[1],
                           oValve => "ST10_Stopper_InterfaceDB".Command[1].Out.oValve,
                           oReleaseCompleted => "ST10_Stopper_InterfaceDB".Command[1].Out.oReleaseCompleted,
                           oReleaseFault => "ST10_Stopper_InterfaceDB".Command[1].Out.oReleaseFault,
                           oReachFault => "ST10_Stopper_InterfaceDB".Command[1].Out.oReachFault,
                           oNotClear => "ST10_Stopper_InterfaceDB".Command[1].Out.oNotClear);
END_REGION

REGION Network 3 (SCL): A-顶升模组-01阻挡气缸
   (*
   REGION 允许释放条件,根据实际完善:顶升下降且线体运行中
       IF "ST10Cylinder".Cy[2].In.HomePositionSensor AND ("ST350_Motor_InterfaceDB".aDev[1].Run OR "Station_Sys".Manual.Mode) THEN//
           "ST350_Stopper_InterfaceDB".Command[2].In.iReleaseClear := True;
       ELSE
           "ST350_Stopper_InterfaceDB".Command[2].In.iReleaseClear := FALSE;
       END_IF;
   END_REGION

   REGION IO_image
       //InPut
       "ST350_Stopper_InterfaceDB".Command[2].In.iSensor := "iWork01PalletDetection";//本站托盘到位
       "ST350_Stopper_InterfaceDB".Command[2].In.iNextSensor := "iWork02PalletDetection";//后站托盘到位
       "ST350_Stopper_InterfaceDB".Command[2].In.iNextValve := "oA-Lifting-02StopperCylinder";//后站挡停输出

       // //OutPut
        "ST10Cylinder".Cy[1].Inout.AutoGoWork:= "ST350_Stopper_InterfaceDB".Command[2].Out.oValve;//本站挡停输出
   END_REGION

   *0
END_REGION

REGION Network 4: #FB_Stopper_Instance[2] A-顶升模组-01阻挡气缸
   RUNG wire#powerrail
      #FB_Stopper_Instance[2](iNextSensor := wire#w1, iSysInface := "Station_Sys".Interface, iSensor := "ST10_Stopper_InterfaceDB".Command[2].In.iSensor, iNextValve := "ST10_Stopper_InterfaceDB".Command[2].In.iNextValve, iPresentDwell := T#0.3s, iNextEmptyDwell := T#8s, iReleaseClear := "ST10_Stopper_InterfaceDB".Command[2].In.iReleaseClear, iReleaseDwell := T#0.3s, iReleaseFaultTimer := T#8s, iReachFaultTimer := T#8s, io_Dev := "ST10_Stopper_InterfaceDB".aDev[2], oValve => "ST10_Stopper_InterfaceDB".Command[2].Out.oValve, oReleaseCompleted => "ST10_Stopper_InterfaceDB".Command[2].Out.oReleaseCompleted, oReleaseFault => "ST10_Stopper_InterfaceDB".Command[2].Out.oReleaseFault, oReachFault => "ST10_Stopper_InterfaceDB".Command[2].Out.oReachFault, oNotClear => "ST10_Stopper_InterfaceDB".Command[2].Out.oNotClear)
   END_RUNG
   RUNG wire#powerrail
      Contact( "ST10_Stopper_InterfaceDB".Command[2].In.iNextSensor )
   END_RUNG wire#w1
   RUNG wire#powerrail
      I_Contact( "ST10Cylinder".Cy[4].In.HomePositionSensor )
   END_RUNG wire#w1
   // the same network as SCL:
   #FB_Stopper_Instance[2](iSysInface := "Station_Sys".Interface,   // "FB_Stopper"
                           iSensor := "ST10_Stopper_InterfaceDB".Command[2].In.iSensor,
                           iNextSensor := "ST10_Stopper_InterfaceDB".Command[2].In.iNextSensor OR NOT "ST10Cylinder".Cy[4].In.HomePositionSensor,
                           iNextValve := "ST10_Stopper_InterfaceDB".Command[2].In.iNextValve,
                           iPresentDwell := T#0.3s,
                           iNextEmptyDwell := T#8s,
                           iReleaseClear := "ST10_Stopper_InterfaceDB".Command[2].In.iReleaseClear,
                           iReleaseDwell := T#0.3s,
                           iReleaseFaultTimer := T#8s,
                           iReachFaultTimer := T#8s,
                           io_Dev := "ST10_Stopper_InterfaceDB".aDev[2],
                           oValve => "ST10_Stopper_InterfaceDB".Command[2].Out.oValve,
                           oReleaseCompleted => "ST10_Stopper_InterfaceDB".Command[2].Out.oReleaseCompleted,
                           oReleaseFault => "ST10_Stopper_InterfaceDB".Command[2].Out.oReleaseFault,
                           oReachFault => "ST10_Stopper_InterfaceDB".Command[2].Out.oReachFault,
                           oNotClear => "ST10_Stopper_InterfaceDB".Command[2].Out.oNotClear);
END_REGION

REGION Network 5 (SCL): A-顶升模组-02阻挡气缸
   //允许释放条件,根据实际完善:顶升下降且线体运行中
   (*

   REGION IOimage
       //InPut
       "ST350_Stopper_InterfaceDB".Command[3].In.iSensor := "iWork02PalletDetection";//本站托盘到位
       "ST350_Stopper_InterfaceDB".Command[3].In.iNextSensor := "iD-LiftingDetection" AND NOT "iD-LiftingINDetection" ;//后站托盘到位

       //替换后站挡停释放信号：升降机在下&顶升下&无料&允许金托盘
       // "ST350_Stopper_InterfaceDB".Command[3].In.iNextValve := ;//后站挡停输出

       // //OutPut
        "ST10Cylinder".Cy[3].Inout.AutoGoWork := "ST350_Stopper_InterfaceDB".Command[3].Out.oValve;//本站挡停输出


   END_REGION

   *)
END_REGION

REGION Network 6: #FB_Stopper_Instance[3] A-顶升模组-02阻挡气缸
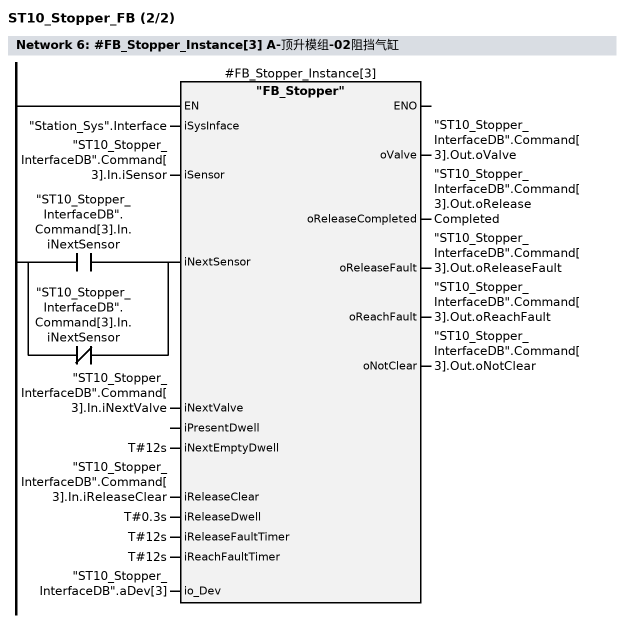
   RUNG wire#powerrail
      #FB_Stopper_Instance[3](iNextSensor := wire#w1, iSysInface := "Station_Sys".Interface, iSensor := "ST10_Stopper_InterfaceDB".Command[3].In.iSensor, iNextValve := "ST10_Stopper_InterfaceDB".Command[3].In.iNextValve, iPresentDwell :=, iNextEmptyDwell := T#12s, iReleaseClear := "ST10_Stopper_InterfaceDB".Command[3].In.iReleaseClear, iReleaseDwell := T#0.3s, iReleaseFaultTimer := T#12s, iReachFaultTimer := T#12s, io_Dev := "ST10_Stopper_InterfaceDB".aDev[3], oValve => "ST10_Stopper_InterfaceDB".Command[3].Out.oValve, oReleaseCompleted => "ST10_Stopper_InterfaceDB".Command[3].Out.oReleaseCompleted, oReleaseFault => "ST10_Stopper_InterfaceDB".Command[3].Out.oReleaseFault, oReachFault => "ST10_Stopper_InterfaceDB".Command[3].Out.oReachFault, oNotClear => "ST10_Stopper_InterfaceDB".Command[3].Out.oNotClear)
   END_RUNG
   RUNG wire#powerrail
      Contact( "ST10_Stopper_InterfaceDB".Command[3].In.iNextSensor )
   END_RUNG wire#w1
   RUNG wire#powerrail
      I_Contact( "ST10_Stopper_InterfaceDB".Command[3].In.iNextSensor )
   END_RUNG wire#w1
   // the same network as SCL:
   #FB_Stopper_Instance[3](iSysInface := "Station_Sys".Interface,   // "FB_Stopper"
                           iSensor := "ST10_Stopper_InterfaceDB".Command[3].In.iSensor,
                           iNextSensor := "ST10_Stopper_InterfaceDB".Command[3].In.iNextSensor OR NOT "ST10_Stopper_InterfaceDB".Command[3].In.iNextSensor,
                           iNextValve := "ST10_Stopper_InterfaceDB".Command[3].In.iNextValve,
                           iNextEmptyDwell := T#12s,
                           iReleaseClear := "ST10_Stopper_InterfaceDB".Command[3].In.iReleaseClear,
                           iReleaseDwell := T#0.3s,
                           iReleaseFaultTimer := T#12s,
                           iReachFaultTimer := T#12s,
                           io_Dev := "ST10_Stopper_InterfaceDB".aDev[3],
                           oValve => "ST10_Stopper_InterfaceDB".Command[3].Out.oValve,
                           oReleaseCompleted => "ST10_Stopper_InterfaceDB".Command[3].Out.oReleaseCompleted,
                           oReleaseFault => "ST10_Stopper_InterfaceDB".Command[3].Out.oReleaseFault,
                           oReachFault => "ST10_Stopper_InterfaceDB".Command[3].Out.oReachFault,
                           oNotClear => "ST10_Stopper_InterfaceDB".Command[3].Out.oNotClear);
END_REGION
END_FUNCTION_BLOCK

FUNCTION_BLOCK "ST10_StopperCtrl"   // FB2601, LAD
TITLE = 输送带控制
{ S7_Optimized_Access := 'FALSE' }
// stored: AutoNumber false, SetENOAutomatically false
   VAR
      Stopper { S7_SetPoint := 'True'} : Array[1..100] of "StopperCtrl";
   END_VAR
   VAR_TEMP   // added for the SCL form of the ladder/FBD networks
      _w1 : Bool;
   END_VAR
BEGIN

REGION Network 1: ------------------------------------------------------------------------------------------------------------------------------ / ------------------------------------------------ H -------------------------------------------------------------------------
END_REGION

REGION Network 2: H-shaftLoadingStopperCylinder1
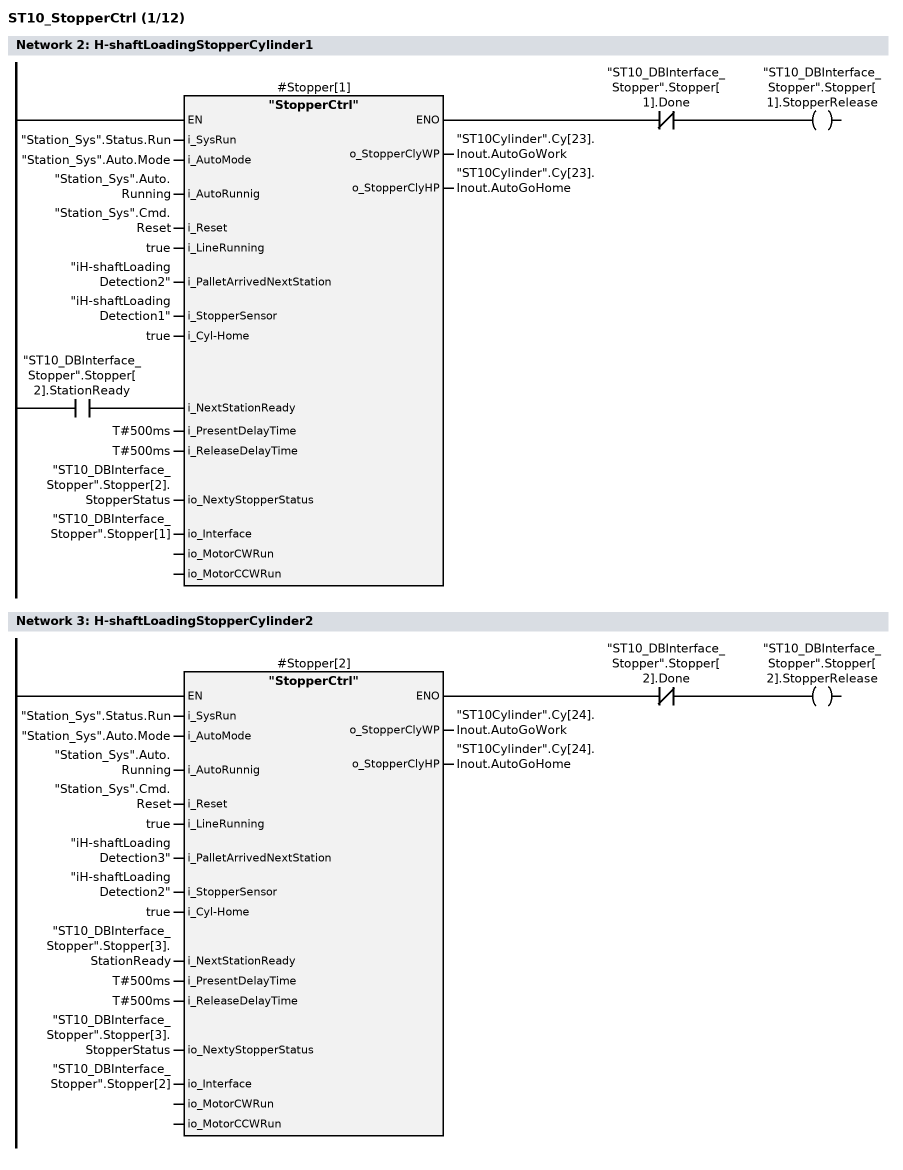
   RUNG wire#powerrail
      #Stopper[1](i_NextStationReady := wire#w1, i_SysRun := "Station_Sys".Status.Run, i_AutoMode := "Station_Sys".Auto.Mode, i_AutoRunnig := "Station_Sys".Auto.Running, i_Reset := "Station_Sys".Cmd.Reset, i_LineRunning := true, i_PalletArrivedNextStation := "iH-shaftLoadingDetection2", i_StopperSensor := "iH-shaftLoadingDetection1", "i_Cyl-Home" := true, i_PresentDelayTime := T#500ms, i_ReleaseDelayTime := T#500ms, io_NextyStopperStatus := "ST10_DBInterface_Stopper".Stopper[2].StopperStatus, io_Interface := "ST10_DBInterface_Stopper".Stopper[1], io_MotorCWRun :=, io_MotorCCWRun :=, o_StopperClyWP => "ST10Cylinder".Cy[23].Inout.AutoGoWork, o_StopperClyHP => "ST10Cylinder".Cy[23].Inout.AutoGoHome)
      I_Contact( "ST10_DBInterface_Stopper".Stopper[1].Done )
      Coil( "ST10_DBInterface_Stopper".Stopper[1].StopperRelease )
   END_RUNG
   RUNG wire#powerrail
      Contact( "ST10_DBInterface_Stopper".Stopper[2].StationReady )
   END_RUNG wire#w1
   // the same network as SCL:
   #Stopper[1](i_SysRun := "Station_Sys".Status.Run,   // "StopperCtrl"
               i_AutoMode := "Station_Sys".Auto.Mode,
               i_AutoRunnig := "Station_Sys".Auto.Running,
               i_Reset := "Station_Sys".Cmd.Reset,
               i_LineRunning := true,
               i_PalletArrivedNextStation := "iH-shaftLoadingDetection2",
               i_StopperSensor := "iH-shaftLoadingDetection1",
               "i_Cyl-Home" := true,
               i_NextStationReady := "ST10_DBInterface_Stopper".Stopper[2].StationReady,
               i_PresentDelayTime := T#500ms,
               i_ReleaseDelayTime := T#500ms,
               io_NextyStopperStatus := "ST10_DBInterface_Stopper".Stopper[2].StopperStatus,
               io_Interface := "ST10_DBInterface_Stopper".Stopper[1],
               o_StopperClyWP => "ST10Cylinder".Cy[23].Inout.AutoGoWork,
               o_StopperClyHP => "ST10Cylinder".Cy[23].Inout.AutoGoHome,
               ENO => #_w1);
   "ST10_DBInterface_Stopper".Stopper[1].StopperRelease := #_w1 AND NOT "ST10_DBInterface_Stopper".Stopper[1].Done;
END_REGION

REGION Network 3: H-shaftLoadingStopperCylinder2
   RUNG wire#powerrail
      #Stopper[2](i_SysRun := "Station_Sys".Status.Run, i_AutoMode := "Station_Sys".Auto.Mode, i_AutoRunnig := "Station_Sys".Auto.Running, i_Reset := "Station_Sys".Cmd.Reset, i_LineRunning := true, i_PalletArrivedNextStation := "iH-shaftLoadingDetection3", i_StopperSensor := "iH-shaftLoadingDetection2", "i_Cyl-Home" := true, i_NextStationReady := "ST10_DBInterface_Stopper".Stopper[3].StationReady, i_PresentDelayTime := T#500ms, i_ReleaseDelayTime := T#500ms, io_NextyStopperStatus := "ST10_DBInterface_Stopper".Stopper[3].StopperStatus, io_Interface := "ST10_DBInterface_Stopper".Stopper[2], io_MotorCWRun :=, io_MotorCCWRun :=, o_StopperClyWP => "ST10Cylinder".Cy[24].Inout.AutoGoWork, o_StopperClyHP => "ST10Cylinder".Cy[24].Inout.AutoGoHome)
      I_Contact( "ST10_DBInterface_Stopper".Stopper[2].Done )
      Coil( "ST10_DBInterface_Stopper".Stopper[2].StopperRelease )
   END_RUNG
   // the same network as SCL:
   #Stopper[2](i_SysRun := "Station_Sys".Status.Run,   // "StopperCtrl"
               i_AutoMode := "Station_Sys".Auto.Mode,
               i_AutoRunnig := "Station_Sys".Auto.Running,
               i_Reset := "Station_Sys".Cmd.Reset,
               i_LineRunning := true,
               i_PalletArrivedNextStation := "iH-shaftLoadingDetection3",
               i_StopperSensor := "iH-shaftLoadingDetection2",
               "i_Cyl-Home" := true,
               i_NextStationReady := "ST10_DBInterface_Stopper".Stopper[3].StationReady,
               i_PresentDelayTime := T#500ms,
               i_ReleaseDelayTime := T#500ms,
               io_NextyStopperStatus := "ST10_DBInterface_Stopper".Stopper[3].StopperStatus,
               io_Interface := "ST10_DBInterface_Stopper".Stopper[2],
               o_StopperClyWP => "ST10Cylinder".Cy[24].Inout.AutoGoWork,
               o_StopperClyHP => "ST10Cylinder".Cy[24].Inout.AutoGoHome,
               ENO => #_w1);
   "ST10_DBInterface_Stopper".Stopper[2].StopperRelease := #_w1 AND NOT "ST10_DBInterface_Stopper".Stopper[2].Done;
END_REGION

REGION Network 4: H-shaftLoadingStopperCylinder3
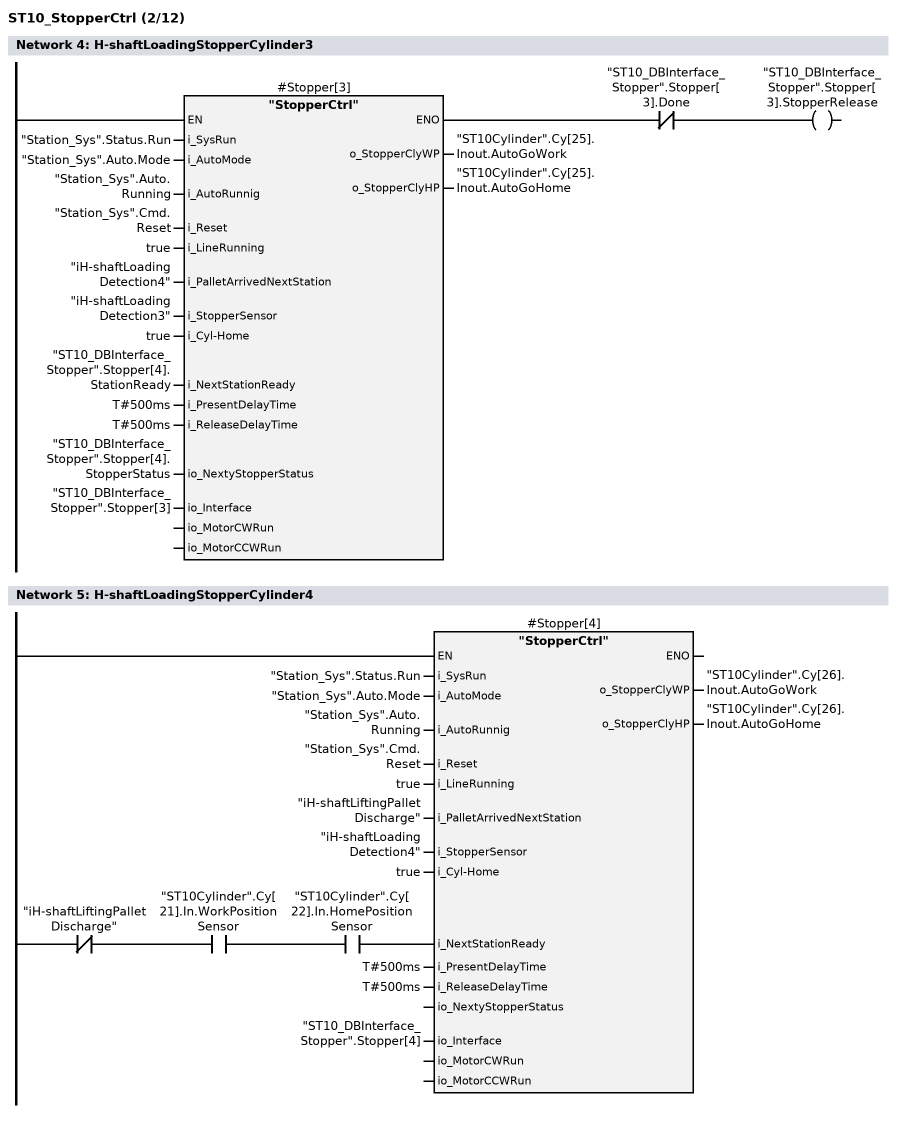
   RUNG wire#powerrail
      #Stopper[3](i_SysRun := "Station_Sys".Status.Run, i_AutoMode := "Station_Sys".Auto.Mode, i_AutoRunnig := "Station_Sys".Auto.Running, i_Reset := "Station_Sys".Cmd.Reset, i_LineRunning := true, i_PalletArrivedNextStation := "iH-shaftLoadingDetection4", i_StopperSensor := "iH-shaftLoadingDetection3", "i_Cyl-Home" := true, i_NextStationReady := "ST10_DBInterface_Stopper".Stopper[4].StationReady, i_PresentDelayTime := T#500ms, i_ReleaseDelayTime := T#500ms, io_NextyStopperStatus := "ST10_DBInterface_Stopper".Stopper[4].StopperStatus, io_Interface := "ST10_DBInterface_Stopper".Stopper[3], io_MotorCWRun :=, io_MotorCCWRun :=, o_StopperClyWP => "ST10Cylinder".Cy[25].Inout.AutoGoWork, o_StopperClyHP => "ST10Cylinder".Cy[25].Inout.AutoGoHome)
      I_Contact( "ST10_DBInterface_Stopper".Stopper[3].Done )
      Coil( "ST10_DBInterface_Stopper".Stopper[3].StopperRelease )
   END_RUNG
   // the same network as SCL:
   #Stopper[3](i_SysRun := "Station_Sys".Status.Run,   // "StopperCtrl"
               i_AutoMode := "Station_Sys".Auto.Mode,
               i_AutoRunnig := "Station_Sys".Auto.Running,
               i_Reset := "Station_Sys".Cmd.Reset,
               i_LineRunning := true,
               i_PalletArrivedNextStation := "iH-shaftLoadingDetection4",
               i_StopperSensor := "iH-shaftLoadingDetection3",
               "i_Cyl-Home" := true,
               i_NextStationReady := "ST10_DBInterface_Stopper".Stopper[4].StationReady,
               i_PresentDelayTime := T#500ms,
               i_ReleaseDelayTime := T#500ms,
               io_NextyStopperStatus := "ST10_DBInterface_Stopper".Stopper[4].StopperStatus,
               io_Interface := "ST10_DBInterface_Stopper".Stopper[3],
               o_StopperClyWP => "ST10Cylinder".Cy[25].Inout.AutoGoWork,
               o_StopperClyHP => "ST10Cylinder".Cy[25].Inout.AutoGoHome,
               ENO => #_w1);
   "ST10_DBInterface_Stopper".Stopper[3].StopperRelease := #_w1 AND NOT "ST10_DBInterface_Stopper".Stopper[3].Done;
END_REGION

REGION Network 5: H-shaftLoadingStopperCylinder4
   RUNG wire#powerrail
      #Stopper[4](i_NextStationReady := wire#w1, i_SysRun := "Station_Sys".Status.Run, i_AutoMode := "Station_Sys".Auto.Mode, i_AutoRunnig := "Station_Sys".Auto.Running, i_Reset := "Station_Sys".Cmd.Reset, i_LineRunning := true, i_PalletArrivedNextStation := "iH-shaftLiftingPalletDischarge", i_StopperSensor := "iH-shaftLoadingDetection4", "i_Cyl-Home" := true, i_PresentDelayTime := T#500ms, i_ReleaseDelayTime := T#500ms, io_NextyStopperStatus :=, io_Interface := "ST10_DBInterface_Stopper".Stopper[4], io_MotorCWRun :=, io_MotorCCWRun :=, o_StopperClyWP => "ST10Cylinder".Cy[26].Inout.AutoGoWork, o_StopperClyHP => "ST10Cylinder".Cy[26].Inout.AutoGoHome)
   END_RUNG
   RUNG wire#powerrail
      I_Contact( "iH-shaftLiftingPalletDischarge" )
      Contact( "ST10Cylinder".Cy[21].In.WorkPositionSensor )
      Contact( "ST10Cylinder".Cy[22].In.HomePositionSensor )
   END_RUNG wire#w1
   // the same network as SCL:
   #Stopper[4](i_SysRun := "Station_Sys".Status.Run,   // "StopperCtrl"
               i_AutoMode := "Station_Sys".Auto.Mode,
               i_AutoRunnig := "Station_Sys".Auto.Running,
               i_Reset := "Station_Sys".Cmd.Reset,
               i_LineRunning := true,
               i_PalletArrivedNextStation := "iH-shaftLiftingPalletDischarge",
               i_StopperSensor := "iH-shaftLoadingDetection4",
               "i_Cyl-Home" := true,
               i_NextStationReady := NOT "iH-shaftLiftingPalletDischarge" AND "ST10Cylinder".Cy[21].In.WorkPositionSensor AND "ST10Cylinder".Cy[22].In.HomePositionSensor,
               i_PresentDelayTime := T#500ms,
               i_ReleaseDelayTime := T#500ms,
               io_Interface := "ST10_DBInterface_Stopper".Stopper[4],
               o_StopperClyWP => "ST10Cylinder".Cy[26].Inout.AutoGoWork,
               o_StopperClyHP => "ST10Cylinder".Cy[26].Inout.AutoGoHome);
END_REGION

REGION Network 6: H-shaftTakeStopperCylinder1
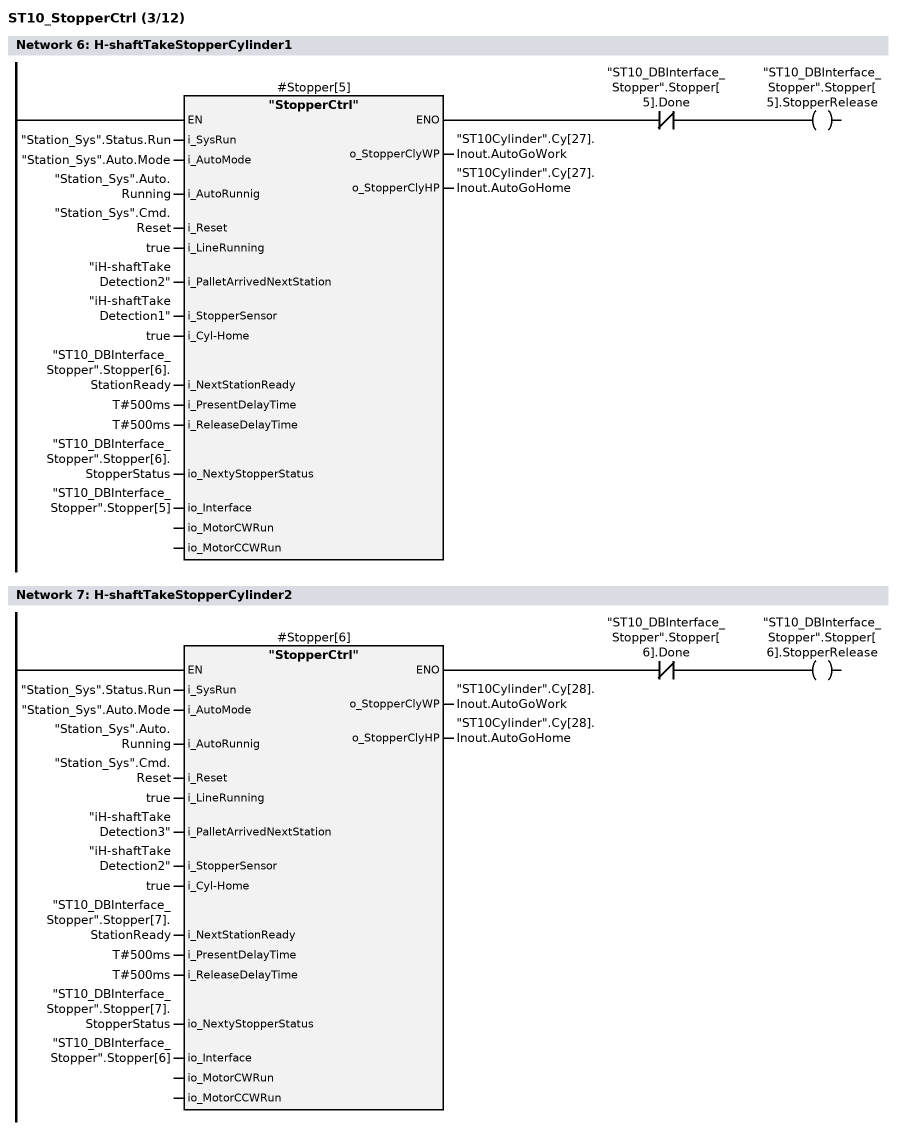
   RUNG wire#powerrail
      #Stopper[5](i_SysRun := "Station_Sys".Status.Run, i_AutoMode := "Station_Sys".Auto.Mode, i_AutoRunnig := "Station_Sys".Auto.Running, i_Reset := "Station_Sys".Cmd.Reset, i_LineRunning := true, i_PalletArrivedNextStation := "iH-shaftTakeDetection2", i_StopperSensor := "iH-shaftTakeDetection1", "i_Cyl-Home" := true, i_NextStationReady := "ST10_DBInterface_Stopper".Stopper[6].StationReady, i_PresentDelayTime := T#500ms, i_ReleaseDelayTime := T#500ms, io_NextyStopperStatus := "ST10_DBInterface_Stopper".Stopper[6].StopperStatus, io_Interface := "ST10_DBInterface_Stopper".Stopper[5], io_MotorCWRun :=, io_MotorCCWRun :=, o_StopperClyWP => "ST10Cylinder".Cy[27].Inout.AutoGoWork, o_StopperClyHP => "ST10Cylinder".Cy[27].Inout.AutoGoHome)
      I_Contact( "ST10_DBInterface_Stopper".Stopper[5].Done )
      Coil( "ST10_DBInterface_Stopper".Stopper[5].StopperRelease )
   END_RUNG
   // the same network as SCL:
   #Stopper[5](i_SysRun := "Station_Sys".Status.Run,   // "StopperCtrl"
               i_AutoMode := "Station_Sys".Auto.Mode,
               i_AutoRunnig := "Station_Sys".Auto.Running,
               i_Reset := "Station_Sys".Cmd.Reset,
               i_LineRunning := true,
               i_PalletArrivedNextStation := "iH-shaftTakeDetection2",
               i_StopperSensor := "iH-shaftTakeDetection1",
               "i_Cyl-Home" := true,
               i_NextStationReady := "ST10_DBInterface_Stopper".Stopper[6].StationReady,
               i_PresentDelayTime := T#500ms,
               i_ReleaseDelayTime := T#500ms,
               io_NextyStopperStatus := "ST10_DBInterface_Stopper".Stopper[6].StopperStatus,
               io_Interface := "ST10_DBInterface_Stopper".Stopper[5],
               o_StopperClyWP => "ST10Cylinder".Cy[27].Inout.AutoGoWork,
               o_StopperClyHP => "ST10Cylinder".Cy[27].Inout.AutoGoHome,
               ENO => #_w1);
   "ST10_DBInterface_Stopper".Stopper[5].StopperRelease := #_w1 AND NOT "ST10_DBInterface_Stopper".Stopper[5].Done;
END_REGION

REGION Network 7: H-shaftTakeStopperCylinder2
   RUNG wire#powerrail
      #Stopper[6](i_SysRun := "Station_Sys".Status.Run, i_AutoMode := "Station_Sys".Auto.Mode, i_AutoRunnig := "Station_Sys".Auto.Running, i_Reset := "Station_Sys".Cmd.Reset, i_LineRunning := true, i_PalletArrivedNextStation := "iH-shaftTakeDetection3", i_StopperSensor := "iH-shaftTakeDetection2", "i_Cyl-Home" := true, i_NextStationReady := "ST10_DBInterface_Stopper".Stopper[7].StationReady, i_PresentDelayTime := T#500ms, i_ReleaseDelayTime := T#500ms, io_NextyStopperStatus := "ST10_DBInterface_Stopper".Stopper[7].StopperStatus, io_Interface := "ST10_DBInterface_Stopper".Stopper[6], io_MotorCWRun :=, io_MotorCCWRun :=, o_StopperClyWP => "ST10Cylinder".Cy[28].Inout.AutoGoWork, o_StopperClyHP => "ST10Cylinder".Cy[28].Inout.AutoGoHome)
      I_Contact( "ST10_DBInterface_Stopper".Stopper[6].Done )
      Coil( "ST10_DBInterface_Stopper".Stopper[6].StopperRelease )
   END_RUNG
   // the same network as SCL:
   #Stopper[6](i_SysRun := "Station_Sys".Status.Run,   // "StopperCtrl"
               i_AutoMode := "Station_Sys".Auto.Mode,
               i_AutoRunnig := "Station_Sys".Auto.Running,
               i_Reset := "Station_Sys".Cmd.Reset,
               i_LineRunning := true,
               i_PalletArrivedNextStation := "iH-shaftTakeDetection3",
               i_StopperSensor := "iH-shaftTakeDetection2",
               "i_Cyl-Home" := true,
               i_NextStationReady := "ST10_DBInterface_Stopper".Stopper[7].StationReady,
               i_PresentDelayTime := T#500ms,
               i_ReleaseDelayTime := T#500ms,
               io_NextyStopperStatus := "ST10_DBInterface_Stopper".Stopper[7].StopperStatus,
               io_Interface := "ST10_DBInterface_Stopper".Stopper[6],
               o_StopperClyWP => "ST10Cylinder".Cy[28].Inout.AutoGoWork,
               o_StopperClyHP => "ST10Cylinder".Cy[28].Inout.AutoGoHome,
               ENO => #_w1);
   "ST10_DBInterface_Stopper".Stopper[6].StopperRelease := #_w1 AND NOT "ST10_DBInterface_Stopper".Stopper[6].Done;
END_REGION

REGION Network 8: H-shaftTakeStopperCylinder3
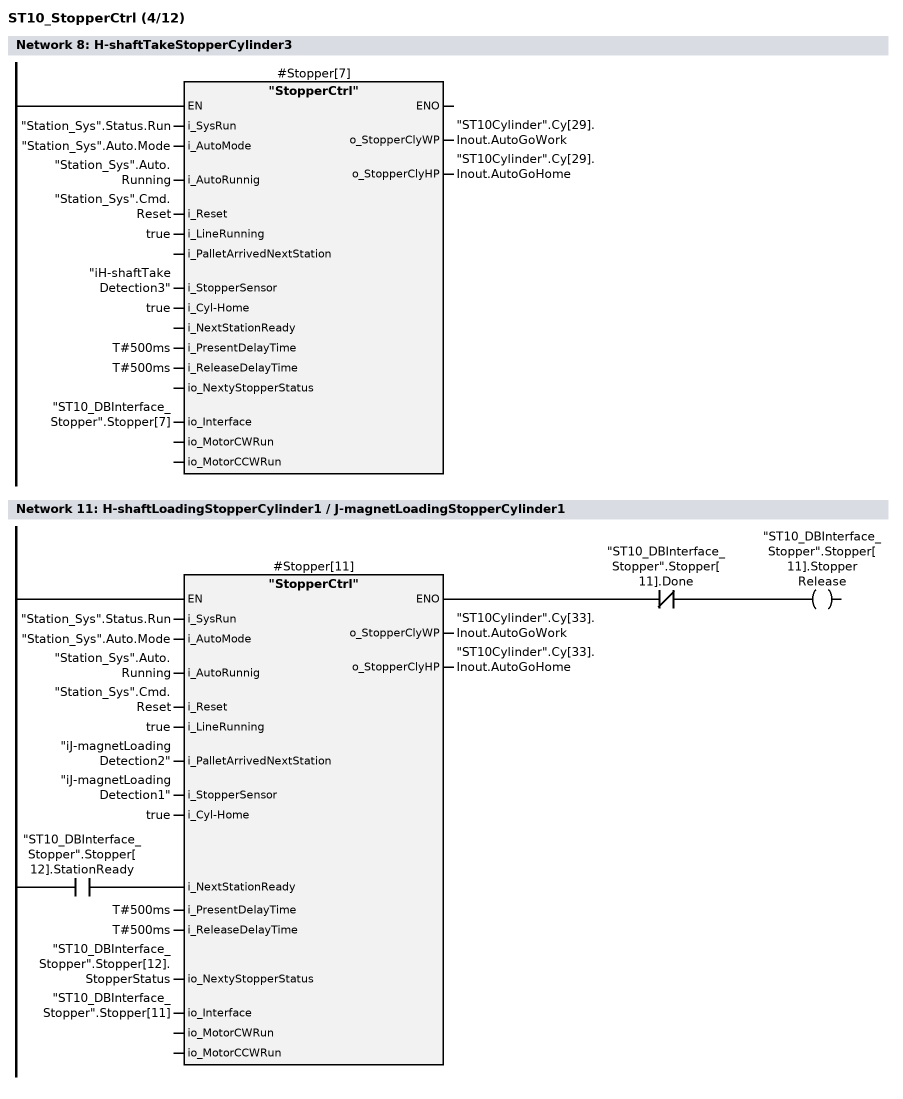
   RUNG wire#powerrail
      #Stopper[7](i_SysRun := "Station_Sys".Status.Run, i_AutoMode := "Station_Sys".Auto.Mode, i_AutoRunnig := "Station_Sys".Auto.Running, i_Reset := "Station_Sys".Cmd.Reset, i_LineRunning := true, i_PalletArrivedNextStation :=, i_StopperSensor := "iH-shaftTakeDetection3", "i_Cyl-Home" := true, i_NextStationReady :=, i_PresentDelayTime := T#500ms, i_ReleaseDelayTime := T#500ms, io_NextyStopperStatus :=, io_Interface := "ST10_DBInterface_Stopper".Stopper[7], io_MotorCWRun :=, io_MotorCCWRun :=, o_StopperClyWP => "ST10Cylinder".Cy[29].Inout.AutoGoWork, o_StopperClyHP => "ST10Cylinder".Cy[29].Inout.AutoGoHome)
   END_RUNG
   // the same network as SCL:
   #Stopper[7](i_SysRun := "Station_Sys".Status.Run,   // "StopperCtrl"
               i_AutoMode := "Station_Sys".Auto.Mode,
               i_AutoRunnig := "Station_Sys".Auto.Running,
               i_Reset := "Station_Sys".Cmd.Reset,
               i_LineRunning := true,
               i_StopperSensor := "iH-shaftTakeDetection3",
               "i_Cyl-Home" := true,
               i_PresentDelayTime := T#500ms,
               i_ReleaseDelayTime := T#500ms,
               io_Interface := "ST10_DBInterface_Stopper".Stopper[7],
               o_StopperClyWP => "ST10Cylinder".Cy[29].Inout.AutoGoWork,
               o_StopperClyHP => "ST10Cylinder".Cy[29].Inout.AutoGoHome);
END_REGION

REGION Network 9: -------------------------------------------------------------------------------------------------------------------------------
END_REGION

REGION Network 10: ------------------------------------------------------------------------------------------------------------------------------ / ------------------------------------------------ J -------------------------------------------------------------------------
END_REGION

REGION Network 11: H-shaftLoadingStopperCylinder1 / J-magnetLoadingStopperCylinder1
   RUNG wire#powerrail
      #Stopper[11](i_NextStationReady := wire#w1, i_SysRun := "Station_Sys".Status.Run, i_AutoMode := "Station_Sys".Auto.Mode, i_AutoRunnig := "Station_Sys".Auto.Running, i_Reset := "Station_Sys".Cmd.Reset, i_LineRunning := true, i_PalletArrivedNextStation := "iJ-magnetLoadingDetection2", i_StopperSensor := "iJ-magnetLoadingDetection1", "i_Cyl-Home" := true, i_PresentDelayTime := T#500ms, i_ReleaseDelayTime := T#500ms, io_NextyStopperStatus := "ST10_DBInterface_Stopper".Stopper[12].StopperStatus, io_Interface := "ST10_DBInterface_Stopper".Stopper[11], io_MotorCWRun :=, io_MotorCCWRun :=, o_StopperClyWP => "ST10Cylinder".Cy[33].Inout.AutoGoWork, o_StopperClyHP => "ST10Cylinder".Cy[33].Inout.AutoGoHome)
      I_Contact( "ST10_DBInterface_Stopper".Stopper[11].Done )
      Coil( "ST10_DBInterface_Stopper".Stopper[11].StopperRelease )
   END_RUNG
   RUNG wire#powerrail
      Contact( "ST10_DBInterface_Stopper".Stopper[12].StationReady )
   END_RUNG wire#w1
   // the same network as SCL:
   #Stopper[11](i_SysRun := "Station_Sys".Status.Run,   // "StopperCtrl"
                i_AutoMode := "Station_Sys".Auto.Mode,
                i_AutoRunnig := "Station_Sys".Auto.Running,
                i_Reset := "Station_Sys".Cmd.Reset,
                i_LineRunning := true,
                i_PalletArrivedNextStation := "iJ-magnetLoadingDetection2",
                i_StopperSensor := "iJ-magnetLoadingDetection1",
                "i_Cyl-Home" := true,
                i_NextStationReady := "ST10_DBInterface_Stopper".Stopper[12].StationReady,
                i_PresentDelayTime := T#500ms,
                i_ReleaseDelayTime := T#500ms,
                io_NextyStopperStatus := "ST10_DBInterface_Stopper".Stopper[12].StopperStatus,
                io_Interface := "ST10_DBInterface_Stopper".Stopper[11],
                o_StopperClyWP => "ST10Cylinder".Cy[33].Inout.AutoGoWork,
                o_StopperClyHP => "ST10Cylinder".Cy[33].Inout.AutoGoHome,
                ENO => #_w1);
   "ST10_DBInterface_Stopper".Stopper[11].StopperRelease := #_w1 AND NOT "ST10_DBInterface_Stopper".Stopper[11].Done;
END_REGION

REGION Network 12: H-shaftLoadingStopperCylinder2 / J-magnetLoadingStopperCylinder2
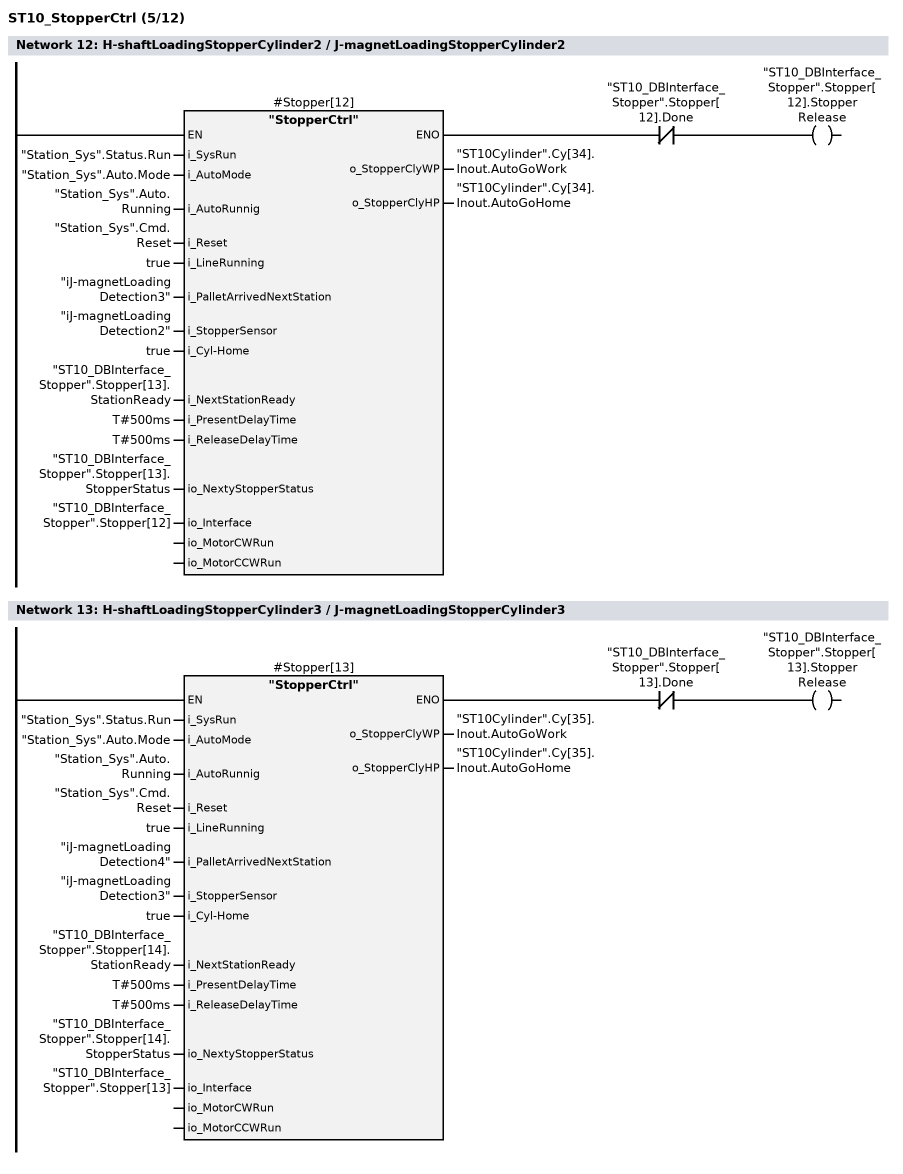
   RUNG wire#powerrail
      #Stopper[12](i_SysRun := "Station_Sys".Status.Run, i_AutoMode := "Station_Sys".Auto.Mode, i_AutoRunnig := "Station_Sys".Auto.Running, i_Reset := "Station_Sys".Cmd.Reset, i_LineRunning := true, i_PalletArrivedNextStation := "iJ-magnetLoadingDetection3", i_StopperSensor := "iJ-magnetLoadingDetection2", "i_Cyl-Home" := true, i_NextStationReady := "ST10_DBInterface_Stopper".Stopper[13].StationReady, i_PresentDelayTime := T#500ms, i_ReleaseDelayTime := T#500ms, io_NextyStopperStatus := "ST10_DBInterface_Stopper".Stopper[13].StopperStatus, io_Interface := "ST10_DBInterface_Stopper".Stopper[12], io_MotorCWRun :=, io_MotorCCWRun :=, o_StopperClyWP => "ST10Cylinder".Cy[34].Inout.AutoGoWork, o_StopperClyHP => "ST10Cylinder".Cy[34].Inout.AutoGoHome)
      I_Contact( "ST10_DBInterface_Stopper".Stopper[12].Done )
      Coil( "ST10_DBInterface_Stopper".Stopper[12].StopperRelease )
   END_RUNG
   // the same network as SCL:
   #Stopper[12](i_SysRun := "Station_Sys".Status.Run,   // "StopperCtrl"
                i_AutoMode := "Station_Sys".Auto.Mode,
                i_AutoRunnig := "Station_Sys".Auto.Running,
                i_Reset := "Station_Sys".Cmd.Reset,
                i_LineRunning := true,
                i_PalletArrivedNextStation := "iJ-magnetLoadingDetection3",
                i_StopperSensor := "iJ-magnetLoadingDetection2",
                "i_Cyl-Home" := true,
                i_NextStationReady := "ST10_DBInterface_Stopper".Stopper[13].StationReady,
                i_PresentDelayTime := T#500ms,
                i_ReleaseDelayTime := T#500ms,
                io_NextyStopperStatus := "ST10_DBInterface_Stopper".Stopper[13].StopperStatus,
                io_Interface := "ST10_DBInterface_Stopper".Stopper[12],
                o_StopperClyWP => "ST10Cylinder".Cy[34].Inout.AutoGoWork,
                o_StopperClyHP => "ST10Cylinder".Cy[34].Inout.AutoGoHome,
                ENO => #_w1);
   "ST10_DBInterface_Stopper".Stopper[12].StopperRelease := #_w1 AND NOT "ST10_DBInterface_Stopper".Stopper[12].Done;
END_REGION

REGION Network 13: H-shaftLoadingStopperCylinder3 / J-magnetLoadingStopperCylinder3
   RUNG wire#powerrail
      #Stopper[13](i_SysRun := "Station_Sys".Status.Run, i_AutoMode := "Station_Sys".Auto.Mode, i_AutoRunnig := "Station_Sys".Auto.Running, i_Reset := "Station_Sys".Cmd.Reset, i_LineRunning := true, i_PalletArrivedNextStation := "iJ-magnetLoadingDetection4", i_StopperSensor := "iJ-magnetLoadingDetection3", "i_Cyl-Home" := true, i_NextStationReady := "ST10_DBInterface_Stopper".Stopper[14].StationReady, i_PresentDelayTime := T#500ms, i_ReleaseDelayTime := T#500ms, io_NextyStopperStatus := "ST10_DBInterface_Stopper".Stopper[14].StopperStatus, io_Interface := "ST10_DBInterface_Stopper".Stopper[13], io_MotorCWRun :=, io_MotorCCWRun :=, o_StopperClyWP => "ST10Cylinder".Cy[35].Inout.AutoGoWork, o_StopperClyHP => "ST10Cylinder".Cy[35].Inout.AutoGoHome)
      I_Contact( "ST10_DBInterface_Stopper".Stopper[13].Done )
      Coil( "ST10_DBInterface_Stopper".Stopper[13].StopperRelease )
   END_RUNG
   // the same network as SCL:
   #Stopper[13](i_SysRun := "Station_Sys".Status.Run,   // "StopperCtrl"
                i_AutoMode := "Station_Sys".Auto.Mode,
                i_AutoRunnig := "Station_Sys".Auto.Running,
                i_Reset := "Station_Sys".Cmd.Reset,
                i_LineRunning := true,
                i_PalletArrivedNextStation := "iJ-magnetLoadingDetection4",
                i_StopperSensor := "iJ-magnetLoadingDetection3",
                "i_Cyl-Home" := true,
                i_NextStationReady := "ST10_DBInterface_Stopper".Stopper[14].StationReady,
                i_PresentDelayTime := T#500ms,
                i_ReleaseDelayTime := T#500ms,
                io_NextyStopperStatus := "ST10_DBInterface_Stopper".Stopper[14].StopperStatus,
                io_Interface := "ST10_DBInterface_Stopper".Stopper[13],
                o_StopperClyWP => "ST10Cylinder".Cy[35].Inout.AutoGoWork,
                o_StopperClyHP => "ST10Cylinder".Cy[35].Inout.AutoGoHome,
                ENO => #_w1);
   "ST10_DBInterface_Stopper".Stopper[13].StopperRelease := #_w1 AND NOT "ST10_DBInterface_Stopper".Stopper[13].Done;
END_REGION

REGION Network 14: H-shaftLoadingStopperCylinder4 / J-magnetLoadingStopperCylinder4
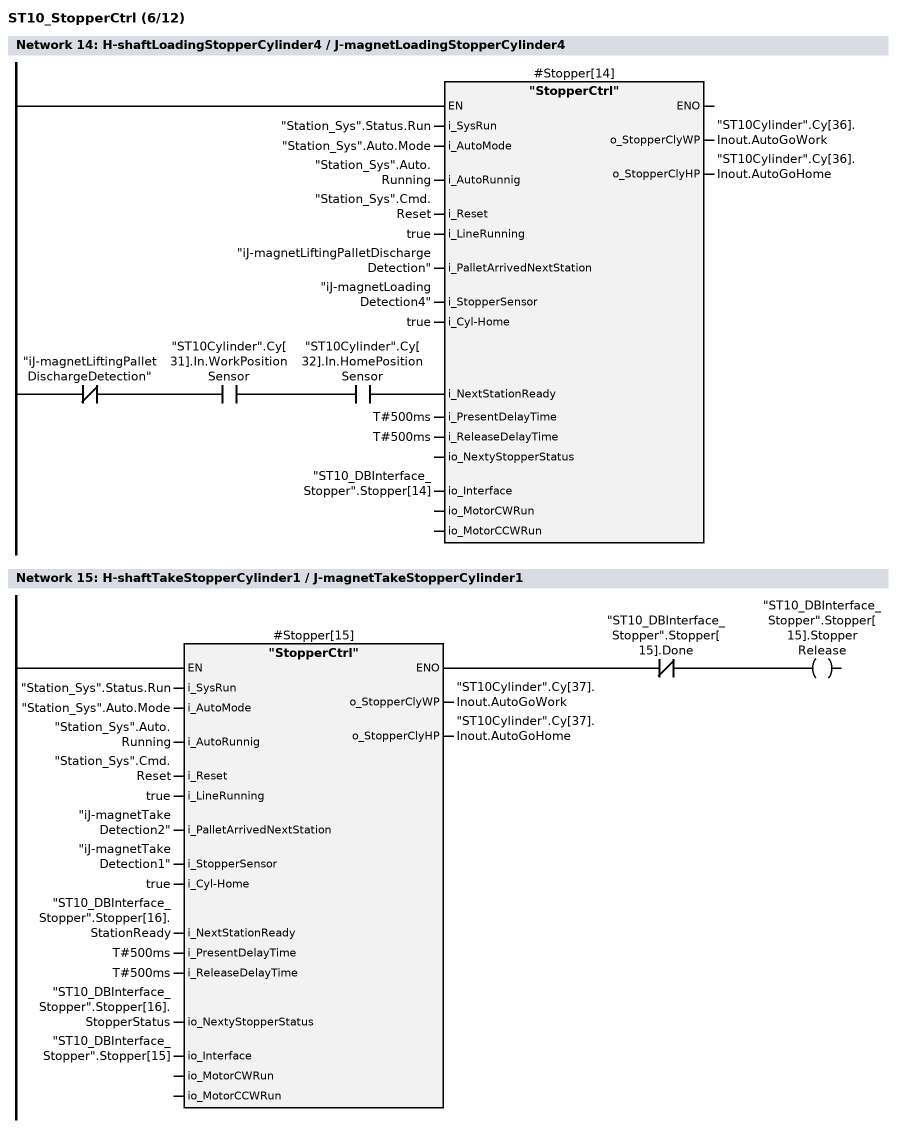
   RUNG wire#powerrail
      #Stopper[14](i_NextStationReady := wire#w1, i_SysRun := "Station_Sys".Status.Run, i_AutoMode := "Station_Sys".Auto.Mode, i_AutoRunnig := "Station_Sys".Auto.Running, i_Reset := "Station_Sys".Cmd.Reset, i_LineRunning := true, i_PalletArrivedNextStation := "iJ-magnetLiftingPalletDischargeDetection", i_StopperSensor := "iJ-magnetLoadingDetection4", "i_Cyl-Home" := true, i_PresentDelayTime := T#500ms, i_ReleaseDelayTime := T#500ms, io_NextyStopperStatus :=, io_Interface := "ST10_DBInterface_Stopper".Stopper[14], io_MotorCWRun :=, io_MotorCCWRun :=, o_StopperClyWP => "ST10Cylinder".Cy[36].Inout.AutoGoWork, o_StopperClyHP => "ST10Cylinder".Cy[36].Inout.AutoGoHome)
   END_RUNG
   RUNG wire#powerrail
      I_Contact( "iJ-magnetLiftingPalletDischargeDetection" )
      Contact( "ST10Cylinder".Cy[31].In.WorkPositionSensor )
      Contact( "ST10Cylinder".Cy[32].In.HomePositionSensor )
   END_RUNG wire#w1
   // the same network as SCL:
   #Stopper[14](i_SysRun := "Station_Sys".Status.Run,   // "StopperCtrl"
                i_AutoMode := "Station_Sys".Auto.Mode,
                i_AutoRunnig := "Station_Sys".Auto.Running,
                i_Reset := "Station_Sys".Cmd.Reset,
                i_LineRunning := true,
                i_PalletArrivedNextStation := "iJ-magnetLiftingPalletDischargeDetection",
                i_StopperSensor := "iJ-magnetLoadingDetection4",
                "i_Cyl-Home" := true,
                i_NextStationReady := NOT "iJ-magnetLiftingPalletDischargeDetection" AND "ST10Cylinder".Cy[31].In.WorkPositionSensor AND "ST10Cylinder".Cy[32].In.HomePositionSensor,
                i_PresentDelayTime := T#500ms,
                i_ReleaseDelayTime := T#500ms,
                io_Interface := "ST10_DBInterface_Stopper".Stopper[14],
                o_StopperClyWP => "ST10Cylinder".Cy[36].Inout.AutoGoWork,
                o_StopperClyHP => "ST10Cylinder".Cy[36].Inout.AutoGoHome);
END_REGION

REGION Network 15: H-shaftTakeStopperCylinder1 / J-magnetTakeStopperCylinder1
   RUNG wire#powerrail
      #Stopper[15](i_SysRun := "Station_Sys".Status.Run, i_AutoMode := "Station_Sys".Auto.Mode, i_AutoRunnig := "Station_Sys".Auto.Running, i_Reset := "Station_Sys".Cmd.Reset, i_LineRunning := true, i_PalletArrivedNextStation := "iJ-magnetTakeDetection2", i_StopperSensor := "iJ-magnetTakeDetection1", "i_Cyl-Home" := true, i_NextStationReady := "ST10_DBInterface_Stopper".Stopper[16].StationReady, i_PresentDelayTime := T#500ms, i_ReleaseDelayTime := T#500ms, io_NextyStopperStatus := "ST10_DBInterface_Stopper".Stopper[16].StopperStatus, io_Interface := "ST10_DBInterface_Stopper".Stopper[15], io_MotorCWRun :=, io_MotorCCWRun :=, o_StopperClyWP => "ST10Cylinder".Cy[37].Inout.AutoGoWork, o_StopperClyHP => "ST10Cylinder".Cy[37].Inout.AutoGoHome)
      I_Contact( "ST10_DBInterface_Stopper".Stopper[15].Done )
      Coil( "ST10_DBInterface_Stopper".Stopper[15].StopperRelease )
   END_RUNG
   // the same network as SCL:
   #Stopper[15](i_SysRun := "Station_Sys".Status.Run,   // "StopperCtrl"
                i_AutoMode := "Station_Sys".Auto.Mode,
                i_AutoRunnig := "Station_Sys".Auto.Running,
                i_Reset := "Station_Sys".Cmd.Reset,
                i_LineRunning := true,
                i_PalletArrivedNextStation := "iJ-magnetTakeDetection2",
                i_StopperSensor := "iJ-magnetTakeDetection1",
                "i_Cyl-Home" := true,
                i_NextStationReady := "ST10_DBInterface_Stopper".Stopper[16].StationReady,
                i_PresentDelayTime := T#500ms,
                i_ReleaseDelayTime := T#500ms,
                io_NextyStopperStatus := "ST10_DBInterface_Stopper".Stopper[16].StopperStatus,
                io_Interface := "ST10_DBInterface_Stopper".Stopper[15],
                o_StopperClyWP => "ST10Cylinder".Cy[37].Inout.AutoGoWork,
                o_StopperClyHP => "ST10Cylinder".Cy[37].Inout.AutoGoHome,
                ENO => #_w1);
   "ST10_DBInterface_Stopper".Stopper[15].StopperRelease := #_w1 AND NOT "ST10_DBInterface_Stopper".Stopper[15].Done;
END_REGION

REGION Network 16: H-shaftTakeStopperCylinder2 / J-magnetTakeStopperCylinder2
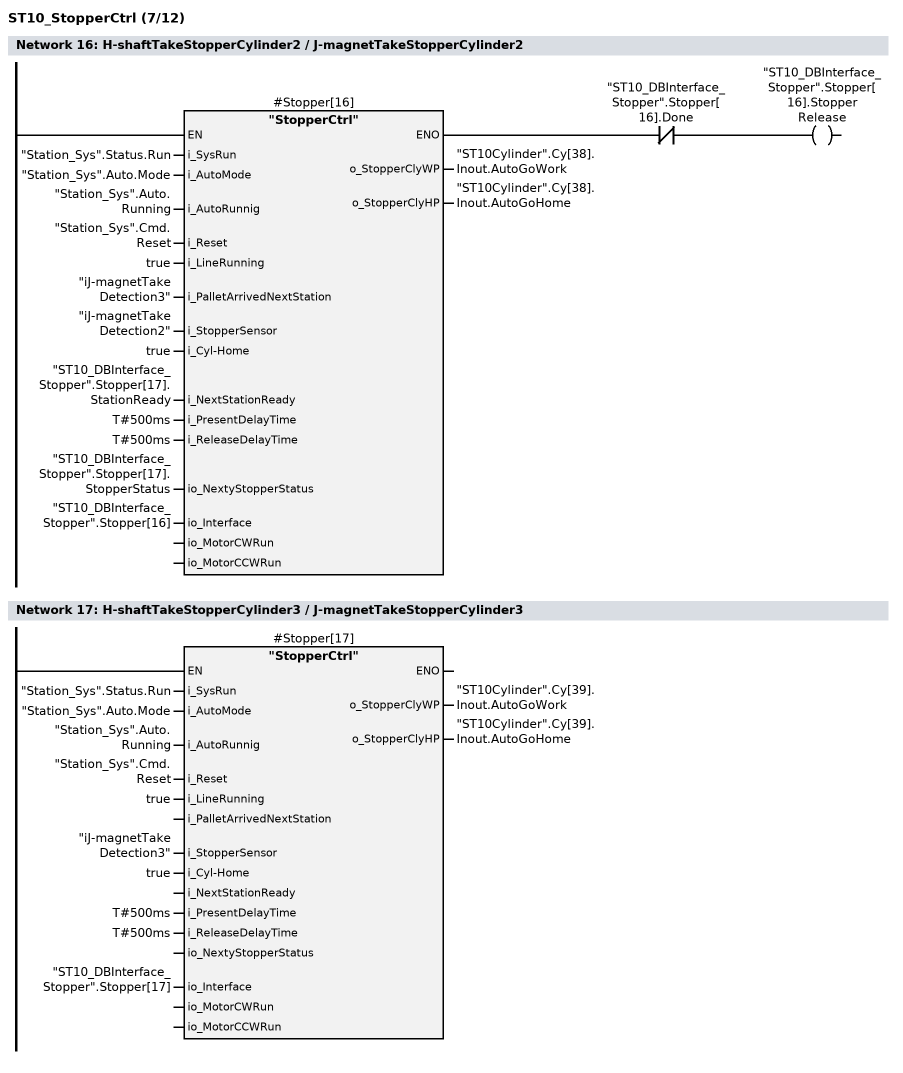
   RUNG wire#powerrail
      #Stopper[16](i_SysRun := "Station_Sys".Status.Run, i_AutoMode := "Station_Sys".Auto.Mode, i_AutoRunnig := "Station_Sys".Auto.Running, i_Reset := "Station_Sys".Cmd.Reset, i_LineRunning := true, i_PalletArrivedNextStation := "iJ-magnetTakeDetection3", i_StopperSensor := "iJ-magnetTakeDetection2", "i_Cyl-Home" := true, i_NextStationReady := "ST10_DBInterface_Stopper".Stopper[17].StationReady, i_PresentDelayTime := T#500ms, i_ReleaseDelayTime := T#500ms, io_NextyStopperStatus := "ST10_DBInterface_Stopper".Stopper[17].StopperStatus, io_Interface := "ST10_DBInterface_Stopper".Stopper[16], io_MotorCWRun :=, io_MotorCCWRun :=, o_StopperClyWP => "ST10Cylinder".Cy[38].Inout.AutoGoWork, o_StopperClyHP => "ST10Cylinder".Cy[38].Inout.AutoGoHome)
      I_Contact( "ST10_DBInterface_Stopper".Stopper[16].Done )
      Coil( "ST10_DBInterface_Stopper".Stopper[16].StopperRelease )
   END_RUNG
   // the same network as SCL:
   #Stopper[16](i_SysRun := "Station_Sys".Status.Run,   // "StopperCtrl"
                i_AutoMode := "Station_Sys".Auto.Mode,
                i_AutoRunnig := "Station_Sys".Auto.Running,
                i_Reset := "Station_Sys".Cmd.Reset,
                i_LineRunning := true,
                i_PalletArrivedNextStation := "iJ-magnetTakeDetection3",
                i_StopperSensor := "iJ-magnetTakeDetection2",
                "i_Cyl-Home" := true,
                i_NextStationReady := "ST10_DBInterface_Stopper".Stopper[17].StationReady,
                i_PresentDelayTime := T#500ms,
                i_ReleaseDelayTime := T#500ms,
                io_NextyStopperStatus := "ST10_DBInterface_Stopper".Stopper[17].StopperStatus,
                io_Interface := "ST10_DBInterface_Stopper".Stopper[16],
                o_StopperClyWP => "ST10Cylinder".Cy[38].Inout.AutoGoWork,
                o_StopperClyHP => "ST10Cylinder".Cy[38].Inout.AutoGoHome,
                ENO => #_w1);
   "ST10_DBInterface_Stopper".Stopper[16].StopperRelease := #_w1 AND NOT "ST10_DBInterface_Stopper".Stopper[16].Done;
END_REGION

REGION Network 17: H-shaftTakeStopperCylinder3 / J-magnetTakeStopperCylinder3
   RUNG wire#powerrail
      #Stopper[17](i_SysRun := "Station_Sys".Status.Run, i_AutoMode := "Station_Sys".Auto.Mode, i_AutoRunnig := "Station_Sys".Auto.Running, i_Reset := "Station_Sys".Cmd.Reset, i_LineRunning := true, i_PalletArrivedNextStation :=, i_StopperSensor := "iJ-magnetTakeDetection3", "i_Cyl-Home" := true, i_NextStationReady :=, i_PresentDelayTime := T#500ms, i_ReleaseDelayTime := T#500ms, io_NextyStopperStatus :=, io_Interface := "ST10_DBInterface_Stopper".Stopper[17], io_MotorCWRun :=, io_MotorCCWRun :=, o_StopperClyWP => "ST10Cylinder".Cy[39].Inout.AutoGoWork, o_StopperClyHP => "ST10Cylinder".Cy[39].Inout.AutoGoHome)
   END_RUNG
   // the same network as SCL:
   #Stopper[17](i_SysRun := "Station_Sys".Status.Run,   // "StopperCtrl"
                i_AutoMode := "Station_Sys".Auto.Mode,
                i_AutoRunnig := "Station_Sys".Auto.Running,
                i_Reset := "Station_Sys".Cmd.Reset,
                i_LineRunning := true,
                i_StopperSensor := "iJ-magnetTakeDetection3",
                "i_Cyl-Home" := true,
                i_PresentDelayTime := T#500ms,
                i_ReleaseDelayTime := T#500ms,
                io_Interface := "ST10_DBInterface_Stopper".Stopper[17],
                o_StopperClyWP => "ST10Cylinder".Cy[39].Inout.AutoGoWork,
                o_StopperClyHP => "ST10Cylinder".Cy[39].Inout.AutoGoHome);
END_REGION

REGION Network 18: -------------------------------------------------------------------------------------------------------------------------------
END_REGION

REGION Network 19: ------------------------------------------------------------------------------------------------------------------------------ / ------------------------------------------------ K -------------------------------------------------------------------------
END_REGION

REGION Network 20: H-shaftLoadingStopperCylinder1 / K-reserveLoadingStopperCylinder1
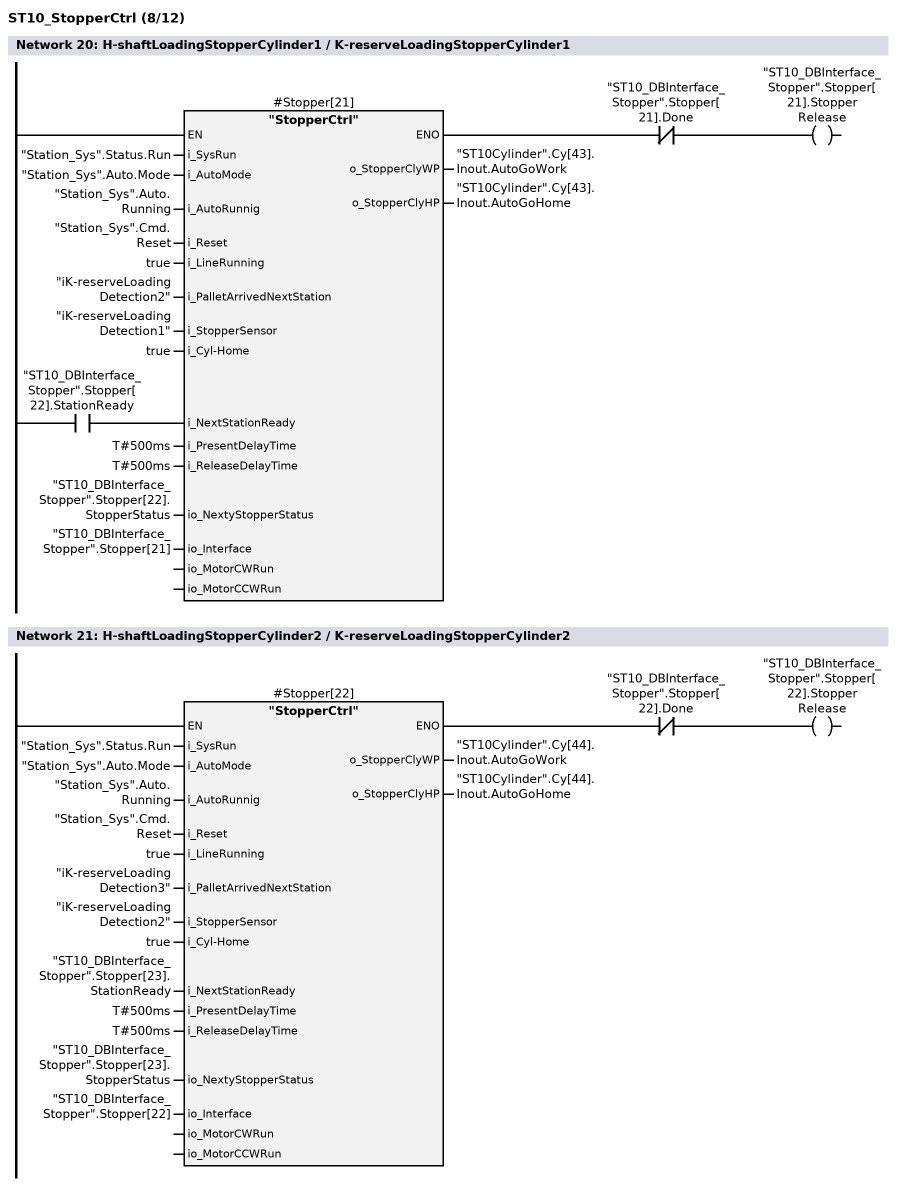
   RUNG wire#powerrail
      #Stopper[21](i_NextStationReady := wire#w1, i_SysRun := "Station_Sys".Status.Run, i_AutoMode := "Station_Sys".Auto.Mode, i_AutoRunnig := "Station_Sys".Auto.Running, i_Reset := "Station_Sys".Cmd.Reset, i_LineRunning := true, i_PalletArrivedNextStation := "iK-reserveLoadingDetection2", i_StopperSensor := "iK-reserveLoadingDetection1", "i_Cyl-Home" := true, i_PresentDelayTime := T#500ms, i_ReleaseDelayTime := T#500ms, io_NextyStopperStatus := "ST10_DBInterface_Stopper".Stopper[22].StopperStatus, io_Interface := "ST10_DBInterface_Stopper".Stopper[21], io_MotorCWRun :=, io_MotorCCWRun :=, o_StopperClyWP => "ST10Cylinder".Cy[43].Inout.AutoGoWork, o_StopperClyHP => "ST10Cylinder".Cy[43].Inout.AutoGoHome)
      I_Contact( "ST10_DBInterface_Stopper".Stopper[21].Done )
      Coil( "ST10_DBInterface_Stopper".Stopper[21].StopperRelease )
   END_RUNG
   RUNG wire#powerrail
      Contact( "ST10_DBInterface_Stopper".Stopper[22].StationReady )
   END_RUNG wire#w1
   // the same network as SCL:
   #Stopper[21](i_SysRun := "Station_Sys".Status.Run,   // "StopperCtrl"
                i_AutoMode := "Station_Sys".Auto.Mode,
                i_AutoRunnig := "Station_Sys".Auto.Running,
                i_Reset := "Station_Sys".Cmd.Reset,
                i_LineRunning := true,
                i_PalletArrivedNextStation := "iK-reserveLoadingDetection2",
                i_StopperSensor := "iK-reserveLoadingDetection1",
                "i_Cyl-Home" := true,
                i_NextStationReady := "ST10_DBInterface_Stopper".Stopper[22].StationReady,
                i_PresentDelayTime := T#500ms,
                i_ReleaseDelayTime := T#500ms,
                io_NextyStopperStatus := "ST10_DBInterface_Stopper".Stopper[22].StopperStatus,
                io_Interface := "ST10_DBInterface_Stopper".Stopper[21],
                o_StopperClyWP => "ST10Cylinder".Cy[43].Inout.AutoGoWork,
                o_StopperClyHP => "ST10Cylinder".Cy[43].Inout.AutoGoHome,
                ENO => #_w1);
   "ST10_DBInterface_Stopper".Stopper[21].StopperRelease := #_w1 AND NOT "ST10_DBInterface_Stopper".Stopper[21].Done;
END_REGION

REGION Network 21: H-shaftLoadingStopperCylinder2 / K-reserveLoadingStopperCylinder2
   RUNG wire#powerrail
      #Stopper[22](i_SysRun := "Station_Sys".Status.Run, i_AutoMode := "Station_Sys".Auto.Mode, i_AutoRunnig := "Station_Sys".Auto.Running, i_Reset := "Station_Sys".Cmd.Reset, i_LineRunning := true, i_PalletArrivedNextStation := "iK-reserveLoadingDetection3", i_StopperSensor := "iK-reserveLoadingDetection2", "i_Cyl-Home" := true, i_NextStationReady := "ST10_DBInterface_Stopper".Stopper[23].StationReady, i_PresentDelayTime := T#500ms, i_ReleaseDelayTime := T#500ms, io_NextyStopperStatus := "ST10_DBInterface_Stopper".Stopper[23].StopperStatus, io_Interface := "ST10_DBInterface_Stopper".Stopper[22], io_MotorCWRun :=, io_MotorCCWRun :=, o_StopperClyWP => "ST10Cylinder".Cy[44].Inout.AutoGoWork, o_StopperClyHP => "ST10Cylinder".Cy[44].Inout.AutoGoHome)
      I_Contact( "ST10_DBInterface_Stopper".Stopper[22].Done )
      Coil( "ST10_DBInterface_Stopper".Stopper[22].StopperRelease )
   END_RUNG
   // the same network as SCL:
   #Stopper[22](i_SysRun := "Station_Sys".Status.Run,   // "StopperCtrl"
                i_AutoMode := "Station_Sys".Auto.Mode,
                i_AutoRunnig := "Station_Sys".Auto.Running,
                i_Reset := "Station_Sys".Cmd.Reset,
                i_LineRunning := true,
                i_PalletArrivedNextStation := "iK-reserveLoadingDetection3",
                i_StopperSensor := "iK-reserveLoadingDetection2",
                "i_Cyl-Home" := true,
                i_NextStationReady := "ST10_DBInterface_Stopper".Stopper[23].StationReady,
                i_PresentDelayTime := T#500ms,
                i_ReleaseDelayTime := T#500ms,
                io_NextyStopperStatus := "ST10_DBInterface_Stopper".Stopper[23].StopperStatus,
                io_Interface := "ST10_DBInterface_Stopper".Stopper[22],
                o_StopperClyWP => "ST10Cylinder".Cy[44].Inout.AutoGoWork,
                o_StopperClyHP => "ST10Cylinder".Cy[44].Inout.AutoGoHome,
                ENO => #_w1);
   "ST10_DBInterface_Stopper".Stopper[22].StopperRelease := #_w1 AND NOT "ST10_DBInterface_Stopper".Stopper[22].Done;
END_REGION

REGION Network 22: H-shaftLoadingStopperCylinder3 / K-reserveLoadingStopperCylinder3
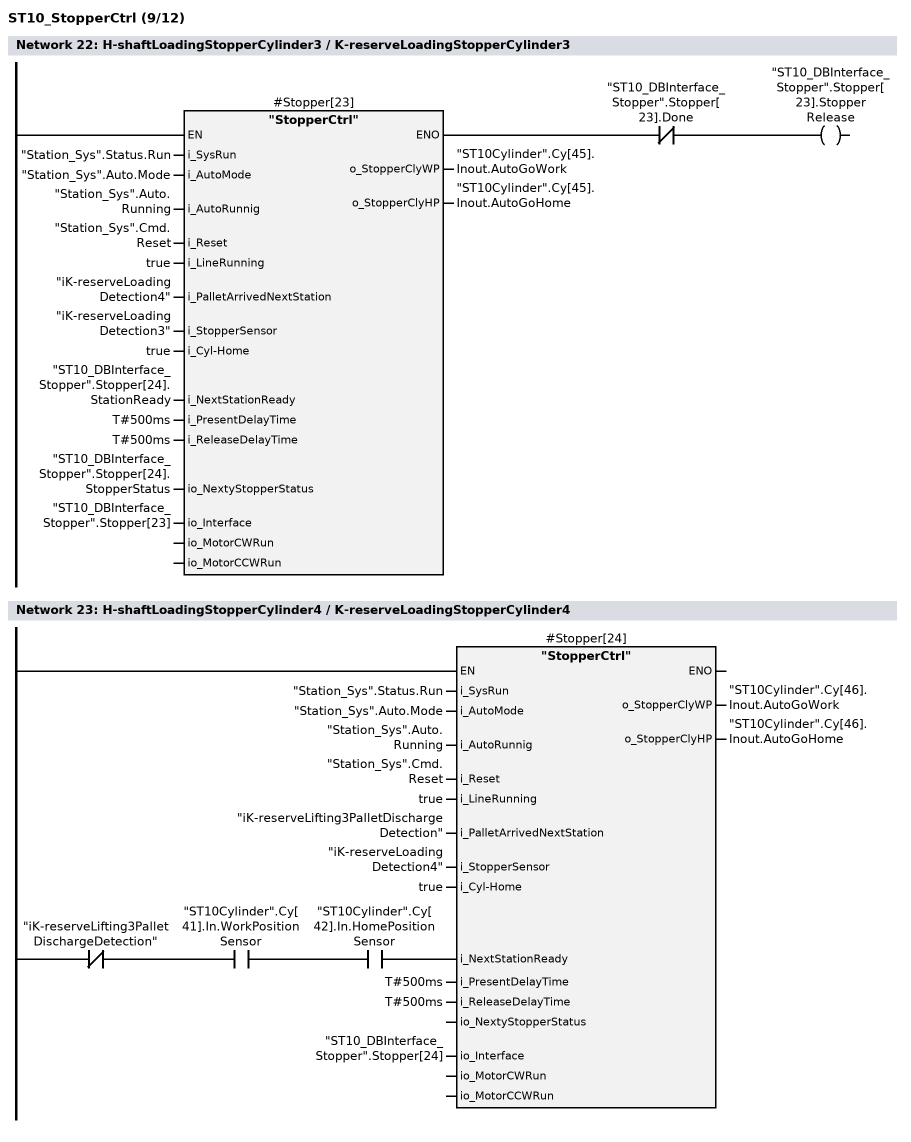
   RUNG wire#powerrail
      #Stopper[23](i_SysRun := "Station_Sys".Status.Run, i_AutoMode := "Station_Sys".Auto.Mode, i_AutoRunnig := "Station_Sys".Auto.Running, i_Reset := "Station_Sys".Cmd.Reset, i_LineRunning := true, i_PalletArrivedNextStation := "iK-reserveLoadingDetection4", i_StopperSensor := "iK-reserveLoadingDetection3", "i_Cyl-Home" := true, i_NextStationReady := "ST10_DBInterface_Stopper".Stopper[24].StationReady, i_PresentDelayTime := T#500ms, i_ReleaseDelayTime := T#500ms, io_NextyStopperStatus := "ST10_DBInterface_Stopper".Stopper[24].StopperStatus, io_Interface := "ST10_DBInterface_Stopper".Stopper[23], io_MotorCWRun :=, io_MotorCCWRun :=, o_StopperClyWP => "ST10Cylinder".Cy[45].Inout.AutoGoWork, o_StopperClyHP => "ST10Cylinder".Cy[45].Inout.AutoGoHome)
      I_Contact( "ST10_DBInterface_Stopper".Stopper[23].Done )
      Coil( "ST10_DBInterface_Stopper".Stopper[23].StopperRelease )
   END_RUNG
   // the same network as SCL:
   #Stopper[23](i_SysRun := "Station_Sys".Status.Run,   // "StopperCtrl"
                i_AutoMode := "Station_Sys".Auto.Mode,
                i_AutoRunnig := "Station_Sys".Auto.Running,
                i_Reset := "Station_Sys".Cmd.Reset,
                i_LineRunning := true,
                i_PalletArrivedNextStation := "iK-reserveLoadingDetection4",
                i_StopperSensor := "iK-reserveLoadingDetection3",
                "i_Cyl-Home" := true,
                i_NextStationReady := "ST10_DBInterface_Stopper".Stopper[24].StationReady,
                i_PresentDelayTime := T#500ms,
                i_ReleaseDelayTime := T#500ms,
                io_NextyStopperStatus := "ST10_DBInterface_Stopper".Stopper[24].StopperStatus,
                io_Interface := "ST10_DBInterface_Stopper".Stopper[23],
                o_StopperClyWP => "ST10Cylinder".Cy[45].Inout.AutoGoWork,
                o_StopperClyHP => "ST10Cylinder".Cy[45].Inout.AutoGoHome,
                ENO => #_w1);
   "ST10_DBInterface_Stopper".Stopper[23].StopperRelease := #_w1 AND NOT "ST10_DBInterface_Stopper".Stopper[23].Done;
END_REGION

REGION Network 23: H-shaftLoadingStopperCylinder4 / K-reserveLoadingStopperCylinder4
   RUNG wire#powerrail
      #Stopper[24](i_NextStationReady := wire#w1, i_SysRun := "Station_Sys".Status.Run, i_AutoMode := "Station_Sys".Auto.Mode, i_AutoRunnig := "Station_Sys".Auto.Running, i_Reset := "Station_Sys".Cmd.Reset, i_LineRunning := true, i_PalletArrivedNextStation := "iK-reserveLifting3PalletDischargeDetection", i_StopperSensor := "iK-reserveLoadingDetection4", "i_Cyl-Home" := true, i_PresentDelayTime := T#500ms, i_ReleaseDelayTime := T#500ms, io_NextyStopperStatus :=, io_Interface := "ST10_DBInterface_Stopper".Stopper[24], io_MotorCWRun :=, io_MotorCCWRun :=, o_StopperClyWP => "ST10Cylinder".Cy[46].Inout.AutoGoWork, o_StopperClyHP => "ST10Cylinder".Cy[46].Inout.AutoGoHome)
   END_RUNG
   RUNG wire#powerrail
      I_Contact( "iK-reserveLifting3PalletDischargeDetection" )
      Contact( "ST10Cylinder".Cy[41].In.WorkPositionSensor )
      Contact( "ST10Cylinder".Cy[42].In.HomePositionSensor )
   END_RUNG wire#w1
   // the same network as SCL:
   #Stopper[24](i_SysRun := "Station_Sys".Status.Run,   // "StopperCtrl"
                i_AutoMode := "Station_Sys".Auto.Mode,
                i_AutoRunnig := "Station_Sys".Auto.Running,
                i_Reset := "Station_Sys".Cmd.Reset,
                i_LineRunning := true,
                i_PalletArrivedNextStation := "iK-reserveLifting3PalletDischargeDetection",
                i_StopperSensor := "iK-reserveLoadingDetection4",
                "i_Cyl-Home" := true,
                i_NextStationReady := NOT "iK-reserveLifting3PalletDischargeDetection" AND "ST10Cylinder".Cy[41].In.WorkPositionSensor AND "ST10Cylinder".Cy[42].In.HomePositionSensor,
                i_PresentDelayTime := T#500ms,
                i_ReleaseDelayTime := T#500ms,
                io_Interface := "ST10_DBInterface_Stopper".Stopper[24],
                o_StopperClyWP => "ST10Cylinder".Cy[46].Inout.AutoGoWork,
                o_StopperClyHP => "ST10Cylinder".Cy[46].Inout.AutoGoHome);
END_REGION

REGION Network 24: H-shaftTakeStopperCylinder1 / K-reserveTakeStopperCylinder1
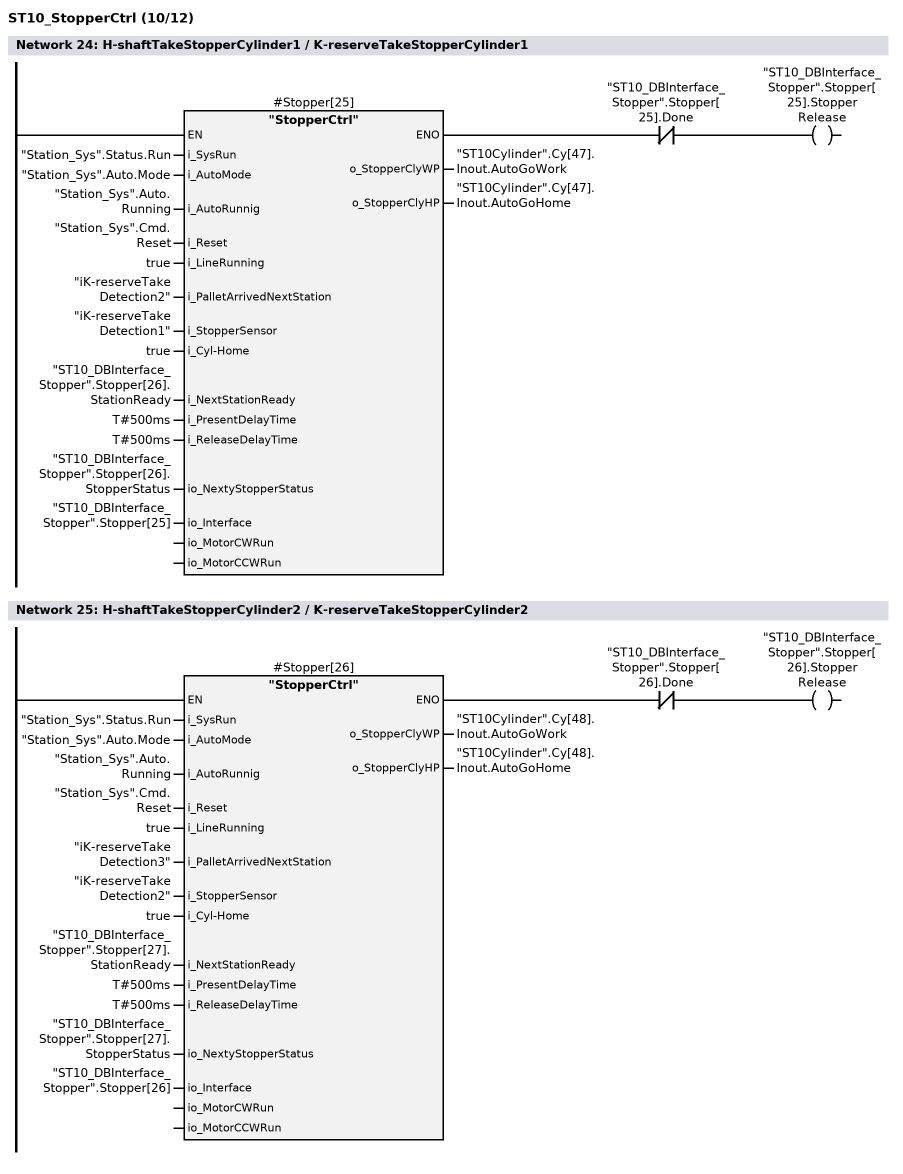
   RUNG wire#powerrail
      #Stopper[25](i_SysRun := "Station_Sys".Status.Run, i_AutoMode := "Station_Sys".Auto.Mode, i_AutoRunnig := "Station_Sys".Auto.Running, i_Reset := "Station_Sys".Cmd.Reset, i_LineRunning := true, i_PalletArrivedNextStation := "iK-reserveTakeDetection2", i_StopperSensor := "iK-reserveTakeDetection1", "i_Cyl-Home" := true, i_NextStationReady := "ST10_DBInterface_Stopper".Stopper[26].StationReady, i_PresentDelayTime := T#500ms, i_ReleaseDelayTime := T#500ms, io_NextyStopperStatus := "ST10_DBInterface_Stopper".Stopper[26].StopperStatus, io_Interface := "ST10_DBInterface_Stopper".Stopper[25], io_MotorCWRun :=, io_MotorCCWRun :=, o_StopperClyWP => "ST10Cylinder".Cy[47].Inout.AutoGoWork, o_StopperClyHP => "ST10Cylinder".Cy[47].Inout.AutoGoHome)
      I_Contact( "ST10_DBInterface_Stopper".Stopper[25].Done )
      Coil( "ST10_DBInterface_Stopper".Stopper[25].StopperRelease )
   END_RUNG
   // the same network as SCL:
   #Stopper[25](i_SysRun := "Station_Sys".Status.Run,   // "StopperCtrl"
                i_AutoMode := "Station_Sys".Auto.Mode,
                i_AutoRunnig := "Station_Sys".Auto.Running,
                i_Reset := "Station_Sys".Cmd.Reset,
                i_LineRunning := true,
                i_PalletArrivedNextStation := "iK-reserveTakeDetection2",
                i_StopperSensor := "iK-reserveTakeDetection1",
                "i_Cyl-Home" := true,
                i_NextStationReady := "ST10_DBInterface_Stopper".Stopper[26].StationReady,
                i_PresentDelayTime := T#500ms,
                i_ReleaseDelayTime := T#500ms,
                io_NextyStopperStatus := "ST10_DBInterface_Stopper".Stopper[26].StopperStatus,
                io_Interface := "ST10_DBInterface_Stopper".Stopper[25],
                o_StopperClyWP => "ST10Cylinder".Cy[47].Inout.AutoGoWork,
                o_StopperClyHP => "ST10Cylinder".Cy[47].Inout.AutoGoHome,
                ENO => #_w1);
   "ST10_DBInterface_Stopper".Stopper[25].StopperRelease := #_w1 AND NOT "ST10_DBInterface_Stopper".Stopper[25].Done;
END_REGION

REGION Network 25: H-shaftTakeStopperCylinder2 / K-reserveTakeStopperCylinder2
   RUNG wire#powerrail
      #Stopper[26](i_SysRun := "Station_Sys".Status.Run, i_AutoMode := "Station_Sys".Auto.Mode, i_AutoRunnig := "Station_Sys".Auto.Running, i_Reset := "Station_Sys".Cmd.Reset, i_LineRunning := true, i_PalletArrivedNextStation := "iK-reserveTakeDetection3", i_StopperSensor := "iK-reserveTakeDetection2", "i_Cyl-Home" := true, i_NextStationReady := "ST10_DBInterface_Stopper".Stopper[27].StationReady, i_PresentDelayTime := T#500ms, i_ReleaseDelayTime := T#500ms, io_NextyStopperStatus := "ST10_DBInterface_Stopper".Stopper[27].StopperStatus, io_Interface := "ST10_DBInterface_Stopper".Stopper[26], io_MotorCWRun :=, io_MotorCCWRun :=, o_StopperClyWP => "ST10Cylinder".Cy[48].Inout.AutoGoWork, o_StopperClyHP => "ST10Cylinder".Cy[48].Inout.AutoGoHome)
      I_Contact( "ST10_DBInterface_Stopper".Stopper[26].Done )
      Coil( "ST10_DBInterface_Stopper".Stopper[26].StopperRelease )
   END_RUNG
   // the same network as SCL:
   #Stopper[26](i_SysRun := "Station_Sys".Status.Run,   // "StopperCtrl"
                i_AutoMode := "Station_Sys".Auto.Mode,
                i_AutoRunnig := "Station_Sys".Auto.Running,
                i_Reset := "Station_Sys".Cmd.Reset,
                i_LineRunning := true,
                i_PalletArrivedNextStation := "iK-reserveTakeDetection3",
                i_StopperSensor := "iK-reserveTakeDetection2",
                "i_Cyl-Home" := true,
                i_NextStationReady := "ST10_DBInterface_Stopper".Stopper[27].StationReady,
                i_PresentDelayTime := T#500ms,
                i_ReleaseDelayTime := T#500ms,
                io_NextyStopperStatus := "ST10_DBInterface_Stopper".Stopper[27].StopperStatus,
                io_Interface := "ST10_DBInterface_Stopper".Stopper[26],
                o_StopperClyWP => "ST10Cylinder".Cy[48].Inout.AutoGoWork,
                o_StopperClyHP => "ST10Cylinder".Cy[48].Inout.AutoGoHome,
                ENO => #_w1);
   "ST10_DBInterface_Stopper".Stopper[26].StopperRelease := #_w1 AND NOT "ST10_DBInterface_Stopper".Stopper[26].Done;
END_REGION

REGION Network 26: H-shaftTakeStopperCylinder3 / K-reserveTakeStopperCylinder3
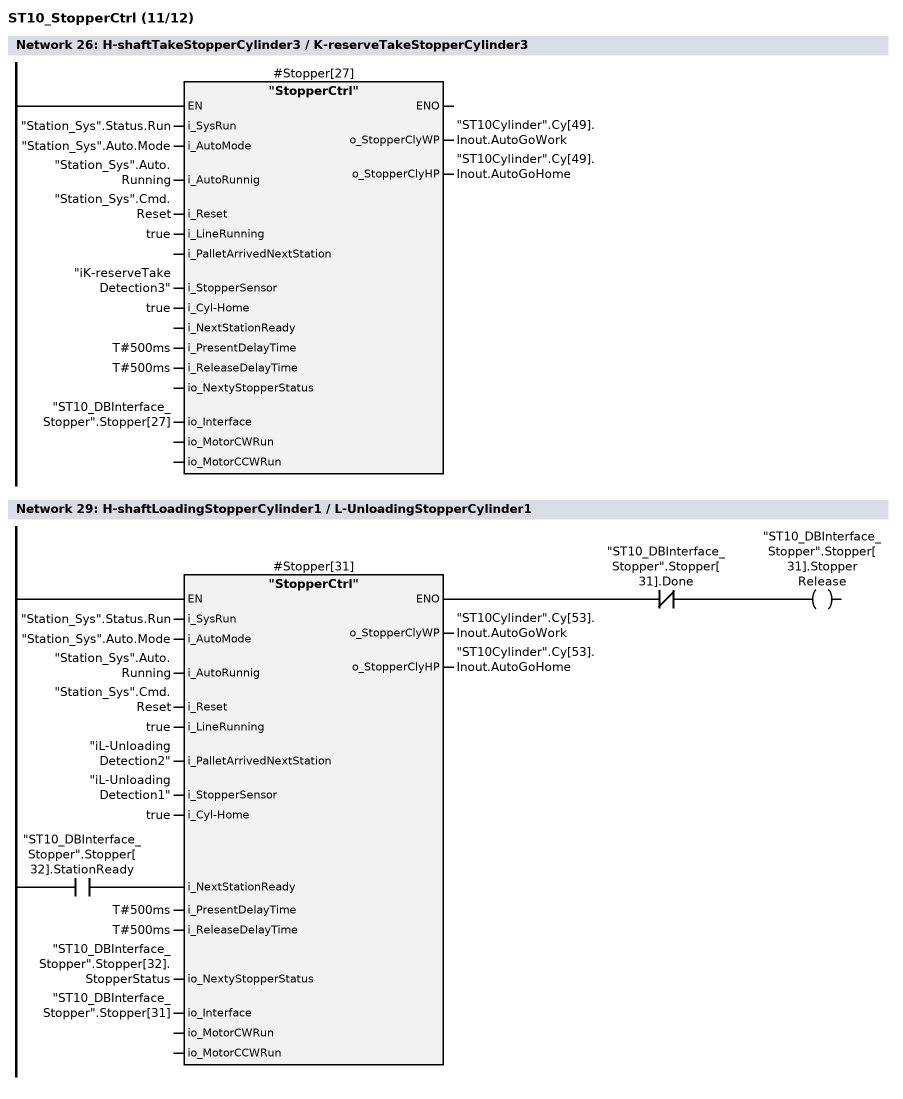
   RUNG wire#powerrail
      #Stopper[27](i_SysRun := "Station_Sys".Status.Run, i_AutoMode := "Station_Sys".Auto.Mode, i_AutoRunnig := "Station_Sys".Auto.Running, i_Reset := "Station_Sys".Cmd.Reset, i_LineRunning := true, i_PalletArrivedNextStation :=, i_StopperSensor := "iK-reserveTakeDetection3", "i_Cyl-Home" := true, i_NextStationReady :=, i_PresentDelayTime := T#500ms, i_ReleaseDelayTime := T#500ms, io_NextyStopperStatus :=, io_Interface := "ST10_DBInterface_Stopper".Stopper[27], io_MotorCWRun :=, io_MotorCCWRun :=, o_StopperClyWP => "ST10Cylinder".Cy[49].Inout.AutoGoWork, o_StopperClyHP => "ST10Cylinder".Cy[49].Inout.AutoGoHome)
   END_RUNG
   // the same network as SCL:
   #Stopper[27](i_SysRun := "Station_Sys".Status.Run,   // "StopperCtrl"
                i_AutoMode := "Station_Sys".Auto.Mode,
                i_AutoRunnig := "Station_Sys".Auto.Running,
                i_Reset := "Station_Sys".Cmd.Reset,
                i_LineRunning := true,
                i_StopperSensor := "iK-reserveTakeDetection3",
                "i_Cyl-Home" := true,
                i_PresentDelayTime := T#500ms,
                i_ReleaseDelayTime := T#500ms,
                io_Interface := "ST10_DBInterface_Stopper".Stopper[27],
                o_StopperClyWP => "ST10Cylinder".Cy[49].Inout.AutoGoWork,
                o_StopperClyHP => "ST10Cylinder".Cy[49].Inout.AutoGoHome);
END_REGION

REGION Network 27: -------------------------------------------------------------------------------------------------------------------------------
END_REGION

REGION Network 28: ------------------------------------------------------------------------------------------------------------------------------ / ------------------------------------------------ L -------------------------------------------------------------------------
END_REGION

REGION Network 29: H-shaftLoadingStopperCylinder1 / L-UnloadingStopperCylinder1
   RUNG wire#powerrail
      #Stopper[31](i_NextStationReady := wire#w1, i_SysRun := "Station_Sys".Status.Run, i_AutoMode := "Station_Sys".Auto.Mode, i_AutoRunnig := "Station_Sys".Auto.Running, i_Reset := "Station_Sys".Cmd.Reset, i_LineRunning := true, i_PalletArrivedNextStation := "iL-UnloadingDetection2", i_StopperSensor := "iL-UnloadingDetection1", "i_Cyl-Home" := true, i_PresentDelayTime := T#500ms, i_ReleaseDelayTime := T#500ms, io_NextyStopperStatus := "ST10_DBInterface_Stopper".Stopper[32].StopperStatus, io_Interface := "ST10_DBInterface_Stopper".Stopper[31], io_MotorCWRun :=, io_MotorCCWRun :=, o_StopperClyWP => "ST10Cylinder".Cy[53].Inout.AutoGoWork, o_StopperClyHP => "ST10Cylinder".Cy[53].Inout.AutoGoHome)
      I_Contact( "ST10_DBInterface_Stopper".Stopper[31].Done )
      Coil( "ST10_DBInterface_Stopper".Stopper[31].StopperRelease )
   END_RUNG
   RUNG wire#powerrail
      Contact( "ST10_DBInterface_Stopper".Stopper[32].StationReady )
   END_RUNG wire#w1
   // the same network as SCL:
   #Stopper[31](i_SysRun := "Station_Sys".Status.Run,   // "StopperCtrl"
                i_AutoMode := "Station_Sys".Auto.Mode,
                i_AutoRunnig := "Station_Sys".Auto.Running,
                i_Reset := "Station_Sys".Cmd.Reset,
                i_LineRunning := true,
                i_PalletArrivedNextStation := "iL-UnloadingDetection2",
                i_StopperSensor := "iL-UnloadingDetection1",
                "i_Cyl-Home" := true,
                i_NextStationReady := "ST10_DBInterface_Stopper".Stopper[32].StationReady,
                i_PresentDelayTime := T#500ms,
                i_ReleaseDelayTime := T#500ms,
                io_NextyStopperStatus := "ST10_DBInterface_Stopper".Stopper[32].StopperStatus,
                io_Interface := "ST10_DBInterface_Stopper".Stopper[31],
                o_StopperClyWP => "ST10Cylinder".Cy[53].Inout.AutoGoWork,
                o_StopperClyHP => "ST10Cylinder".Cy[53].Inout.AutoGoHome,
                ENO => #_w1);
   "ST10_DBInterface_Stopper".Stopper[31].StopperRelease := #_w1 AND NOT "ST10_DBInterface_Stopper".Stopper[31].Done;
END_REGION

REGION Network 30: H-shaftLoadingStopperCylinder2 / L-UnloadingStopperCylinder2
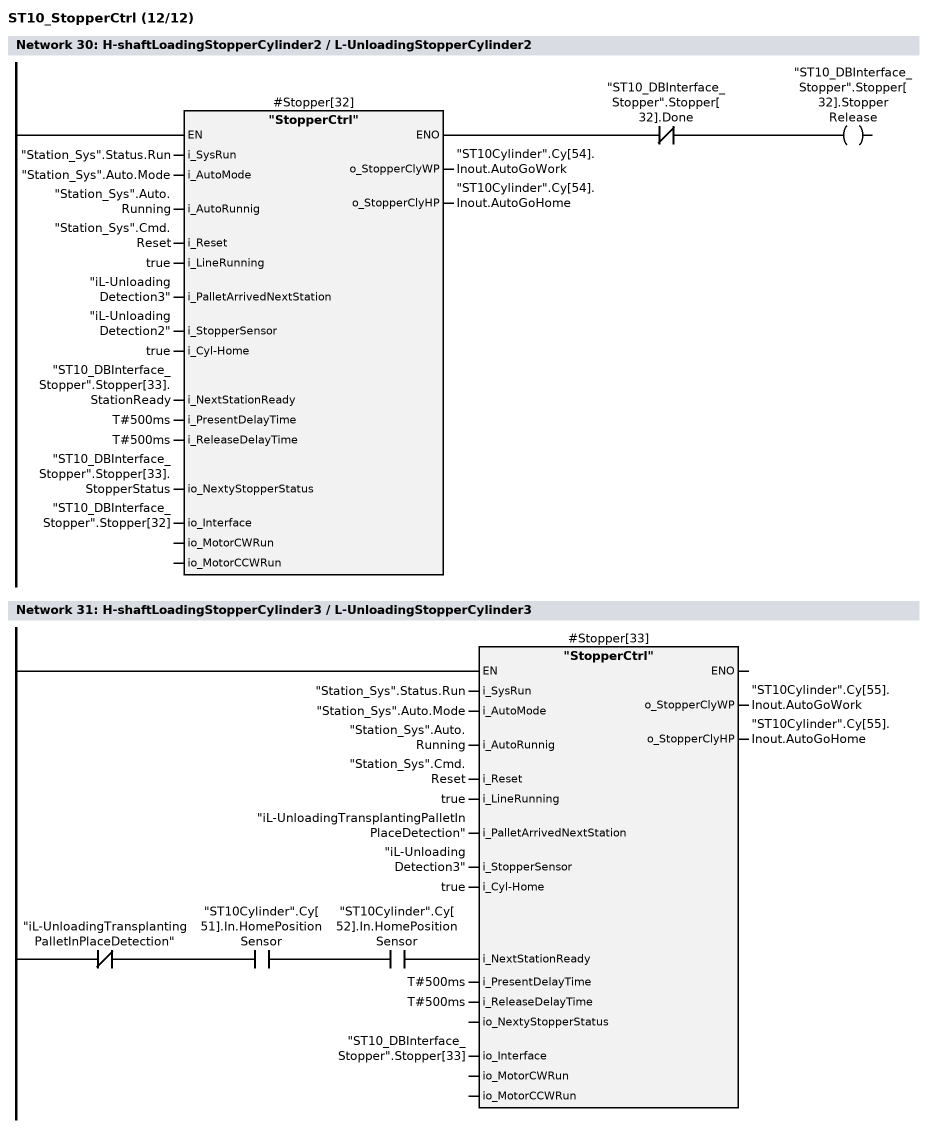
   RUNG wire#powerrail
      #Stopper[32](i_SysRun := "Station_Sys".Status.Run, i_AutoMode := "Station_Sys".Auto.Mode, i_AutoRunnig := "Station_Sys".Auto.Running, i_Reset := "Station_Sys".Cmd.Reset, i_LineRunning := true, i_PalletArrivedNextStation := "iL-UnloadingDetection3", i_StopperSensor := "iL-UnloadingDetection2", "i_Cyl-Home" := true, i_NextStationReady := "ST10_DBInterface_Stopper".Stopper[33].StationReady, i_PresentDelayTime := T#500ms, i_ReleaseDelayTime := T#500ms, io_NextyStopperStatus := "ST10_DBInterface_Stopper".Stopper[33].StopperStatus, io_Interface := "ST10_DBInterface_Stopper".Stopper[32], io_MotorCWRun :=, io_MotorCCWRun :=, o_StopperClyWP => "ST10Cylinder".Cy[54].Inout.AutoGoWork, o_StopperClyHP => "ST10Cylinder".Cy[54].Inout.AutoGoHome)
      I_Contact( "ST10_DBInterface_Stopper".Stopper[32].Done )
      Coil( "ST10_DBInterface_Stopper".Stopper[32].StopperRelease )
   END_RUNG
   // the same network as SCL:
   #Stopper[32](i_SysRun := "Station_Sys".Status.Run,   // "StopperCtrl"
                i_AutoMode := "Station_Sys".Auto.Mode,
                i_AutoRunnig := "Station_Sys".Auto.Running,
                i_Reset := "Station_Sys".Cmd.Reset,
                i_LineRunning := true,
                i_PalletArrivedNextStation := "iL-UnloadingDetection3",
                i_StopperSensor := "iL-UnloadingDetection2",
                "i_Cyl-Home" := true,
                i_NextStationReady := "ST10_DBInterface_Stopper".Stopper[33].StationReady,
                i_PresentDelayTime := T#500ms,
                i_ReleaseDelayTime := T#500ms,
                io_NextyStopperStatus := "ST10_DBInterface_Stopper".Stopper[33].StopperStatus,
                io_Interface := "ST10_DBInterface_Stopper".Stopper[32],
                o_StopperClyWP => "ST10Cylinder".Cy[54].Inout.AutoGoWork,
                o_StopperClyHP => "ST10Cylinder".Cy[54].Inout.AutoGoHome,
                ENO => #_w1);
   "ST10_DBInterface_Stopper".Stopper[32].StopperRelease := #_w1 AND NOT "ST10_DBInterface_Stopper".Stopper[32].Done;
END_REGION

REGION Network 31: H-shaftLoadingStopperCylinder3 / L-UnloadingStopperCylinder3
   RUNG wire#powerrail
      #Stopper[33](i_NextStationReady := wire#w1, i_SysRun := "Station_Sys".Status.Run, i_AutoMode := "Station_Sys".Auto.Mode, i_AutoRunnig := "Station_Sys".Auto.Running, i_Reset := "Station_Sys".Cmd.Reset, i_LineRunning := true, i_PalletArrivedNextStation := "iL-UnloadingTransplantingPalletInPlaceDetection", i_StopperSensor := "iL-UnloadingDetection3", "i_Cyl-Home" := true, i_PresentDelayTime := T#500ms, i_ReleaseDelayTime := T#500ms, io_NextyStopperStatus :=, io_Interface := "ST10_DBInterface_Stopper".Stopper[33], io_MotorCWRun :=, io_MotorCCWRun :=, o_StopperClyWP => "ST10Cylinder".Cy[55].Inout.AutoGoWork, o_StopperClyHP => "ST10Cylinder".Cy[55].Inout.AutoGoHome)
   END_RUNG
   RUNG wire#powerrail
      I_Contact( "iL-UnloadingTransplantingPalletInPlaceDetection" )
      Contact( "ST10Cylinder".Cy[51].In.HomePositionSensor )
      Contact( "ST10Cylinder".Cy[52].In.HomePositionSensor )
   END_RUNG wire#w1
   // the same network as SCL:
   #Stopper[33](i_SysRun := "Station_Sys".Status.Run,   // "StopperCtrl"
                i_AutoMode := "Station_Sys".Auto.Mode,
                i_AutoRunnig := "Station_Sys".Auto.Running,
                i_Reset := "Station_Sys".Cmd.Reset,
                i_LineRunning := true,
                i_PalletArrivedNextStation := "iL-UnloadingTransplantingPalletInPlaceDetection",
                i_StopperSensor := "iL-UnloadingDetection3",
                "i_Cyl-Home" := true,
                i_NextStationReady := NOT "iL-UnloadingTransplantingPalletInPlaceDetection" AND "ST10Cylinder".Cy[51].In.HomePositionSensor AND "ST10Cylinder".Cy[52].In.HomePositionSensor,
                i_PresentDelayTime := T#500ms,
                i_ReleaseDelayTime := T#500ms,
                io_Interface := "ST10_DBInterface_Stopper".Stopper[33],
                o_StopperClyWP => "ST10Cylinder".Cy[55].Inout.AutoGoWork,
                o_StopperClyHP => "ST10Cylinder".Cy[55].Inout.AutoGoHome);
END_REGION

REGION Network 32: -------------------------------------------------------------------------------------------------------------------------------
END_REGION
END_FUNCTION_BLOCK

FUNCTION_BLOCK "StopperCtrl"   // FB2600, LAD
TITLE = stopper program
{ S7_Optimized_Access := 'TRUE' }
// stored: AutoNumber false, MemoryReserve 100, SetENOAutomatically false
   VAR_INPUT
      i_SysRun : Bool;
      i_AutoMode : Bool;
      i_AutoRunnig : Bool;
      i_Reset : Bool;
      i_LineRunning : Bool;
      i_PalletArrivedNextStation : Bool;
      i_StopperSensor : Bool;   // local arrived sensor
      "i_Cyl-Home" : Bool;   // 顶升气缸原始位
      i_NextStationReady : Bool;
      i_PresentDelayTime : Time;
      i_ReleaseDelayTime : Time;
   END_VAR
   VAR_OUTPUT
      o_StopperClyWP : Bool;   // Stopper cylinder
      o_StopperClyHP : Bool;
   END_VAR
   VAR_IN_OUT
      io_NextyStopperStatus : Int;
      io_Interface : "UDT_StopperInterface";
      io_MotorCWRun : Bool;
      io_MotorCCWRun : Bool;
   END_VAR
   VAR RETAIN
      s_Sequence : Int;   // pulse flag
   END_VAR
   VAR
      s_SequenceEnable : Bool;
      s_SequenceFirstEnable : Bool;
      s_StopperSensorOnDelay { S7_SetPoint := 'True'} : TON_TIME;
      s_StopperSensorOffDelay { S7_SetPoint := 'True'} : TON_TIME;
      s_PalletMissingConfirmDelay { S7_SetPoint := 'True'} : TON_TIME;
      s_PalletToNextStationDelay { S7_SetPoint := 'True'} : TON_TIME;
      s_SequenceFirstAutoDelay { S7_SetPoint := 'True'} : TON_TIME;
      s_SequenceFirstAuto { S7_SetPoint := 'True'} : Int;
      s_StopperSensor : Bool;
      s_PalletArrivedNextStation : Bool;
      P : Array[0..10] of Bool;
   END_VAR
   VAR_TEMP
      t_AlwaysOn : Bool;
   END_VAR
   VAR_TEMP   // added for the SCL form of the ladder/FBD networks
      _w1 : Bool;
      _w2 : Bool;
      _w3 : Bool;
      _w4 : Bool;
   END_VAR
BEGIN

REGION Network 1: Always On
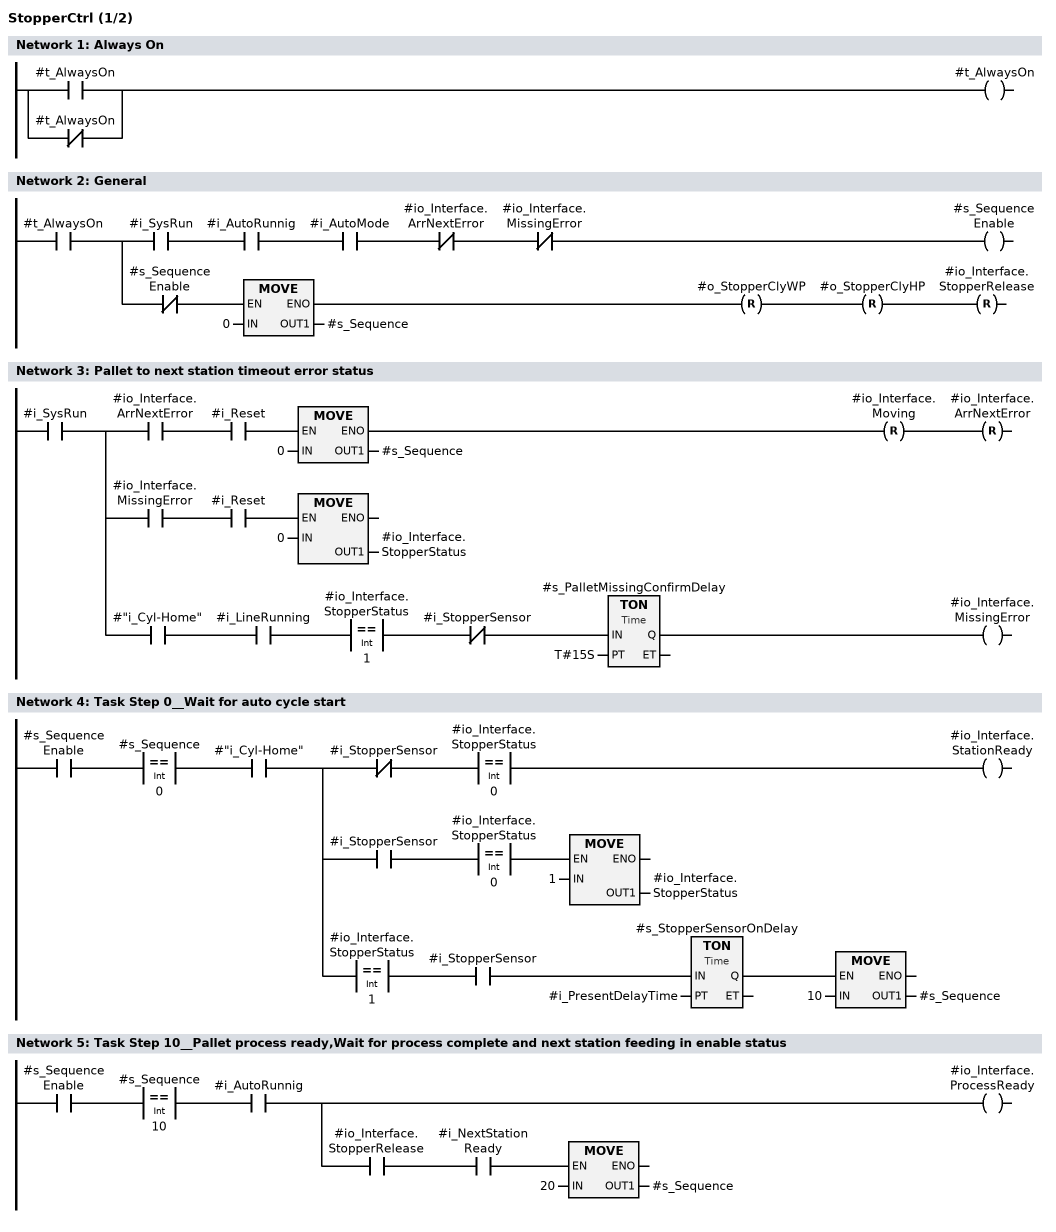
   RUNG wire#powerrail
      Contact( #t_AlwaysOn )
      wire#w1
      Coil( #t_AlwaysOn )
   END_RUNG
   RUNG wire#powerrail
      I_Contact( #t_AlwaysOn )
   END_RUNG wire#w1
   // the same network as SCL:
   #t_AlwaysOn := #t_AlwaysOn OR NOT #t_AlwaysOn;
END_REGION

